// TwinCAT 3 PLC project plc_project
// ProgramVersion: 3.1.4026.24
// libraries:
//   Tc2_Standard, * (Beckhoff Automation GmbH)
//   Tc2_System, * (Beckhoff Automation GmbH)
//   Tc3_Module, * (Beckhoff Automation GmbH)
// project tree:
//   / PlcTask.TcTTO
//   samples/ E_Sample_LargeEnum.TcDUT (not stored), F_Sample_ScaleColorValue.TcPOU (not stored), FB_Sample_AutonomousWarehouseFleetManager.TcPOU, FB_Sample_BatchRecipeExecutionEngine.TcPOU, FB_Sample_DataRingBuffer.TcPOU, FB_Sample_HighDensityDataAnalyticsLogger.TcPOU, FB_Sample_MultiAxisMotionCoordinator.TcPOU (not stored), FB_Sample_MultiStageProcessSupervisor.TcPOU, FB_Sample_StateMachineController.TcPOU (not stored), FB_Sample_ValueBase.TcPOU (not stored), FB_Sample_WidgetBase.TcPOU, GVL_Sample_ParamInflux.TcGVL, GVL_Sample_ShadingConfig.TcGVL (not stored), I_Sample_WidgetInterface.TcIO, ST_Sample_DiagnosticsStruct.TcDUT
//   syntax/ E_Syntax_ExhaustiveComments.TcDUT, E_Syntax_ExplicitIntTyped.TcDUT (not stored), E_Syntax_Flags.TcDUT (not stored), E_Syntax_MultilineAligned.TcDUT (not stored), E_Syntax_TypedExplicit.TcDUT, F_3Args.TcPOU (not stored), F_4Args.TcPOU (not stored), F_5Args.TcPOU (not stored), F_Syntax_Add.TcPOU, F_Syntax_GenericAny.TcPOU, F_Syntax_Return.TcPOU, FB_Syntax_AbstractBase.TcPOU, FB_Syntax_Action.TcPOU (not stored), FB_Syntax_AdvancedSystemExtensions.TcPOU, FB_Syntax_AllVarTypes.TcPOU (not stored), FB_Syntax_AssignAlignmentHeuristics.TcPOU, FB_Syntax_AttributesComprehensive.TcPOU, FB_Syntax_BitAccess.TcPOU, FB_Syntax_Calls.TcPOU (not stored), FB_Syntax_CaseRanges.TcPOU, FB_Syntax_ComplexExpressions.TcPOU, FB_Syntax_ComplexInits.TcPOU, FB_Syntax_ComprehensiveVarBlocks.TcPOU (not stored), FB_Syntax_ConditionalCompile.TcPOU (not stored), FB_Syntax_ControlFlow.TcPOU (not stored), FB_Syntax_DeepControlFlow.TcPOU (not stored), FB_Syntax_DeepNesting.TcPOU, FB_Syntax_Derived.TcPOU, FB_Syntax_DisableRegions.TcPOU (not stored), FB_Syntax_DynamicMem.TcPOU, FB_Syntax_Exceptions.TcPOU (not stored), FB_Syntax_ExhaustiveArraysAndFBInit.TcPOU (not stored), FB_Syntax_ExhaustiveComments.TcPOU, FB_Syntax_ExhaustiveEdgeCases.TcPOU (not stored), FB_Syntax_ExhaustivePragmas.TcPOU (not stored), FB_Syntax_Expressions.TcPOU (not stored), FB_Syntax_ExST.TcPOU, FB_Syntax_FBInitMethods.TcPOU, FB_Syntax_Final.TcPOU (not stored), FB_Syntax_IfMultilineCalls.TcPOU, FB_Syntax_LargeServicePOU.TcPOU, FB_Syntax_LoopControl.TcPOU, FB_Syntax_MathOperators.TcPOU, FB_Syntax_MultiDimArraysAndInits.TcPOU, FB_Syntax_MultiInterfaceDevice.TcPOU (not stored), FB_Syntax_NestedLogCall.TcPOU, FB_Syntax_OOP.TcPOU, FB_Syntax_Pragmas.TcPOU, FB_Syntax_PragmasAndRegions.TcPOU (not stored), FB_Syntax_PropertiesFull.TcPOU, FB_Syntax_PropertySet.TcPOU, FB_Syntax_QueryInterface.TcPOU, FB_Syntax_StringLiterals.TcPOU (not stored), FB_Syntax_StweepDisable.TcPOU, FB_Syntax_SuperThis.TcPOU, FB_Syntax_TimeDate.TcPOU (not stored), FB_Syntax_VarBlocks.TcPOU (not stored), FB_Syntax_VarInOut.TcPOU, FB_Syntax_WrapCallsComprehensive.TcPOU (not stored), FB_Syntax_WrapLongCall.TcPOU, FindAndReplace.TcPOU (not stored), GVL_Syntax_Address.TcGVL, GVL_Syntax_Config.TcGVL (not stored), GVL_Syntax_Global.TcGVL (not stored), GVL_Syntax_Literals.TcGVL, I_Syntax_AdvancedDevice.TcIO (not stored), I_Syntax_BaseDevice.TcIO (not stored), I_Syntax_ExhaustiveComments.TcIO, I_Syntax_Extended.TcIO, I_Syntax_Widget.TcIO (not stored), MAIN.TcPOU, PRG_Syntax_Main.TcPOU, ST_Syntax_Bitfields.TcDUT (not stored), ST_Syntax_ComplexTree.TcDUT (not stored), ST_Syntax_DeepNested.TcDUT (not stored), ST_Syntax_Derived.TcDUT, ST_Syntax_DirectAddressing.TcDUT, ST_Syntax_Dyn.TcDUT (not stored), ST_Syntax_ExhaustiveArrays.TcDUT, ST_Syntax_ExhaustiveComments.TcDUT, ST_Syntax_Mini.TcDUT (not stored), ST_Syntax_PointerRef.TcDUT, T_Syntax_ArraysMultiDim.TcDUT (not stored), T_Syntax_SubrangeEdgeCases.TcDUT, T_Syntax_Types.TcDUT, U_Syntax_ExhaustiveComments.TcDUT, U_Syntax_MultiWordUnion.TcDUT, U_Syntax_Union.TcDUT (not stored)
// real-time tasks:
//   TASK PlcTask: cycle T#10ms, priority 20, ADS port 350

CONFIGURATION plc_project
    RESOURCE PLC ON TwinCAT3
        TASK PlcTask(INTERVAL := T#10ms, PRIORITY := 20);
        PROGRAM MAIN WITH PlcTask : MAIN;
    END_RESOURCE
END_CONFIGURATION

// ---- samples/ST_Sample_DiagnosticsStruct.TcDUT
TYPE ST_Sample_DiagnosticsStruct :
    STRUCT
        (* --- Light device aggregation (previous cycle snapshot) --- *)
        nLightCount                 : UINT; (* Number of reporting light devices *)
        fArtificialLevelSum         : REAL; (* [0..100] - Sum of artificial light levels *)
        fArtificialLevelMean        : REAL; (* [0..100] - Mean artificial light level; 0 if nLightCount = 0 *)
        nLightManualCount           : UINT; (* Number of reporting lights in ManualOperation *)
        nLightExternalOverrideCount : UINT; (* Lights with active prio neither None nor DaylightAutomation *)
        bLightExternalOverride      : BOOL; (* TRUE when nLightExternalOverrideCount > 0 *)
        nLightForeignLightCount     : UINT; (* Of those, the ones actually emitting light (level > 0) *)
        bLightForeignLightActive    : BOOL; (* TRUE when nLightForeignLightCount > 0 *)
        nLightCalibrationCount      : UINT; (* Lights owned by DeskCal this cycle *)

        (* Color temperature aggregation (ColorTemp-capable lights only) *)
        nLightColorTempCount      : UINT; (* Lights reporting a valid color temperature *)
        fLightColorTempKelvinSum  : REAL; (* [K] - Sum of reported color temperatures *)
        fLightColorTempKelvinMean : REAL; (* [K] - Mean color temperature; 0 if nLightColorTempCount = 0 *)

        (* --- Blind device aggregation (previous cycle snapshot) --- *)
        nBlindCount            : UINT; (* Number of reporting blind devices *)
        fBlindPositionSum      : REAL; (* [0..100] - Sum of blind positions *)
        fBlindPositionMean     : REAL; (* [0..100] - Mean blind position; 0 if nBlindCount = 0 *)
        nBlindManualCount      : UINT; (* Number of reporting blinds in ManualOperation *)
        nBlindCalibrationCount : UINT; (* Blinds owned by DeskCal (excl. windows) *)

        (* Angle aggregation (Shade/Sunblind only) *)
        nBlindAngleCount : UINT; (* Blinds reporting a valid angle *)
        fBlindAngleSum   : REAL; (* [deg] - Sum of reported angles *)
        fBlindAngleMean  : REAL; (* [deg] - Mean angle; 0 if nBlindAngleCount = 0 *)

        (* Per NESW facade: 0=North, 1=East, 2=South, 3=West *)
        arrFacadeBlindCount            : ARRAY[0..3] OF UINT; (* Reporting blinds that set this facade bit *)
        arrFacadeBlindPositionMean     : ARRAY[0..3] OF REAL; (* [0..100] - Mean position for that facade bit *)
        arrFacadeBlindCalibrationCount : ARRAY[0..3] OF UINT; (* NESW blinds owned by DeskCal *)
        arrFacadeBlindAngleCount       : ARRAY[0..3] OF UINT; (* Blinds reporting angle for this facade bit *)
        arrFacadeBlindAngleMean        : ARRAY[0..3] OF REAL; (* [deg] - Mean angle for that facade bit *)

        (* --- Occupancy / room sensors (resolved values; *Valid = real source) --- *)
        bMotionSensor              : BOOL; (* Raw motion (sensor or fallback) *)
        bMotionSensorValid         : BOOL; (* TRUE when motion came from stMeasurements *)
        fBrightnessSensorLux       : REAL; (* [Lux] - Effective ceiling / room brightness *)
        bBrightnessSensorValid     : BOOL; (* TRUE when brightness came from stMeasurements *)
        fDeskBrightnessSensorLux   : REAL; (* [Lux] - Effective desk / workplace sensor *)
        bDeskBrightnessSensorValid : BOOL; (* TRUE when desk brightness came from stMeasurements *)
        fHumiditySensor            : REAL; (* [%RH] - Effective room humidity *)
        bHumiditySensorValid       : BOOL; (* TRUE when humidity came from stMeasurements *)
        fCO2Sensor                 : REAL; (* [ppm] - Effective room CO2 / CO2-equivalent *)
        bCO2SensorValid            : BOOL; (* TRUE when CO2 came from stMeasurements *)
        fTemperatureSensor         : REAL; (* [°C] - Effective room temperature *)
        bTemperatureSensorValid    : BOOL; (* TRUE when temperature came from sensor *)
        bOccupancyActive           : BOOL; (* Occupancy: motion hold + Presence delay chains *)
        bOccupancyValid            : BOOL; (* TRUE when occupancy is based on a valid motion sensor *)
    END_STRUCT
END_TYPE

// ---- syntax/E_Syntax_ExhaustiveComments.TcDUT
(*******************************************************************************
 * Enum: E_Syntax_ExhaustiveComments
 * Description: Enumeration with comments on every member and section.
 *******************************************************************************)
TYPE E_Syntax_ExhaustiveComments : (
        // --- Initial / Off states ---
        Uninitialized := 0,  (* System not yet configured *)
        Idle          := 10, // System ready and waiting

        // --- Operational states ---
        Starting := 20, (* Ramping up *)
        Running  := 30, // Normal continuous operation
        Pausing  := 40, (* Transitioning to paused *)
        Paused   := 50, // Temporarily suspended

        // --- Error / Abort states ---
        Stopping      := 80, (* Graceful shutdown *)
        Error         := 90, // Fault detected
        EmergencyStop := 99  (* Immediate safety halt *)
    ) INT;
END_TYPE

// ---- syntax/E_Syntax_TypedExplicit.TcDUT
{attribute 'qualified_only'}
{attribute 'strict'}
TYPE E_Syntax_TypedExplicit : (
        Idle       := 0,   // Initial state
        Starting   := 10,  // Starting sequence
        Running    := 100, // Active processing
        Stopping   := 200, // Ramp down
        ErrorState := -1   // Fault occurred
    ) DINT := Idle;
END_TYPE

// ---- syntax/ST_Syntax_Derived.TcDUT
TYPE ST_Syntax_Derived EXTENDS ST_Syntax_Mini :
    STRUCT
        fExtendedValue : LREAL      := 3.14159;
        sDescription   : STRING(80) := 'Derived Struct';
        bDerivedActive : BOOL;
    END_STRUCT
END_TYPE

// ---- syntax/ST_Syntax_DirectAddressing.TcDUT
TYPE ST_Syntax_DirectAddressing :
    STRUCT
        bInSafetyDoor AT %I* : BOOL;
        nInPosition   AT %I* : INT;
        bOutMotorOn   AT %Q* : BOOL;
        nOutSpeed     AT %Q* : WORD;
        nMemoryStatus AT %M* : DWORD;
    END_STRUCT
END_TYPE

// ---- syntax/ST_Syntax_ExhaustiveArrays.TcDUT
TYPE ST_Syntax_ExhaustiveArrays :
    STRUCT
        arrStaticInts   : ARRAY[1..8] OF INT := [1, 2, 3, 4, 5, 6, 7, 8];
        arrMultiDimInt  : ARRAY[1..2, 1..2] OF INT;
        arrMultilineInt : ARRAY[1..4] OF INT := [
            1, 2,
            3, 4
        ];
        arrNestedMini   : ARRAY[1..2] OF ST_Syntax_Mini := [
            (nId := 1, bActive := TRUE, sName := 'SubA'),
            (nId := 2, bActive := FALSE, sName := 'SubB')
        ];
    END_STRUCT
END_TYPE

// ---- syntax/ST_Syntax_ExhaustiveComments.TcDUT
(*******************************************************************************
 * Struct: ST_Syntax_ExhaustiveComments
 * Description: Data structure with comments in all possible positions.
 *******************************************************************************)
TYPE ST_Syntax_ExhaustiveComments :
    STRUCT
        // --- Identification ---
    nId      : DINT       := 1;      (* Unique device ID *)
        sTag : STRING(31) := 'MAIN'; // System tag name

        // --- Configuration ---
    bEnabled      : BOOL := TRUE;  (* Master enable *)
        fMinLimit : REAL := 0.0;   // Lower threshold
        fMaxLimit : REAL := 100.0; (* Upper threshold *)

        // --- Complex / Nested fields ---
    arrThreshold : ARRAY[1..3] OF REAL := [
        10.0, (* stage 1 *)
        50.0, (* stage 2 *)
        90.0  (* stage 3 *)
    ]; // Multi-stage limits
    END_STRUCT
END_TYPE

// ---- syntax/ST_Syntax_PointerRef.TcDUT
TYPE ST_Syntax_PointerRef :
    STRUCT
        pData : POINTER TO INT;
        rItem : REFERENCE TO INT;
    END_STRUCT
END_TYPE

// ---- syntax/T_Syntax_SubrangeEdgeCases.TcDUT
TYPE T_Syntax_SubrangeEdgeCases : INT(1..100) := 50;

END_TYPE

// ---- syntax/T_Syntax_Types.TcDUT
TYPE T_Syntax_Types :
    STRUCT
        nSubrange   : INT(0..100) := 50;
        aMatrix     : ARRAY[1..3, 1..3] OF REAL;
        sCustomText : STRING(255);
    END_STRUCT
END_TYPE

// ---- syntax/U_Syntax_ExhaustiveComments.TcDUT
(*******************************************************************************
 * Union: U_Syntax_ExhaustiveComments
 * Description: Union testing comments on fields.
 *******************************************************************************)
TYPE U_Syntax_ExhaustiveComments : UNION
        nRawDword : DWORD;               (* 32-bit raw register value *)
        arrBytes  : ARRAY[0..3] OF BYTE; // 4-byte byte access
        arrWords  : ARRAY[0..1] OF WORD; (* 2-word word access *)
    END_UNION
END_TYPE

// ---- syntax/U_Syntax_MultiWordUnion.TcDUT
TYPE U_Syntax_MultiWordUnion : UNION
        nLWord    : LWORD;
        arrDWords : ARRAY[0..1] OF DWORD;
        arrWords  : ARRAY[0..3] OF WORD;
        arrBytes  : ARRAY[0..7] OF BYTE;
    END_UNION
END_TYPE

// ---- samples/GVL_Sample_ParamInflux.TcGVL
{attribute 'qualified_only'}
VAR_GLOBAL CONSTANT
    sDefaultOrg            : STRING(80) := 'ElektroBeckhoff';
    sDefaultBucket         : STRING(80) := 'Telemetry';
    cnMaxBatchSize         : UDINT      := 500;
    cnMaxRetries           : UINT       := 3;
    tDefaultFlushInterval  : TIME       := T#5S;
    tDefaultRequestTimeout : TIME       := T#10S;
END_VAR

// ---- syntax/GVL_Syntax_Address.TcGVL
VAR_GLOBAL
    bInput    AT %I0.0 : BOOL;
    nAnalog   AT %I2   : INT;
    bOutput   AT %Q0.0 : BOOL;
    nSetpoint AT %Q4   : DINT;
END_VAR

// ---- syntax/GVL_Syntax_Literals.TcGVL
VAR_GLOBAL
    todClock           : TOD  := TOD#19:00:00;
    dtEvent            : DT   := DT#2024-01-15-12:30:00;
    nTyped             : DINT := DINT#42;
    nAux, nAux2, nAux3 : UDINT;
END_VAR

// ---- samples/I_Sample_WidgetInterface.TcIO
INTERFACE I_Sample_WidgetInterface EXTENDS __SYSTEM.IQueryInterface

PROPERTY AdsPath : STRING(255)
GET
END_GET
END_PROPERTY

PROPERTY AttributeVariable1 : STRING(80)
GET
END_GET
SET
END_SET
END_PROPERTY

METHOD BuildAttributes : UDINT
VAR_INPUT
    nFlags : DWORD;
END_VAR
END_METHOD

METHOD ProcessCommand : BOOL
VAR_INPUT
    nCommandId : DINT;
    fValue     : LREAL;
END_VAR
VAR_OUTPUT
    bHandled : BOOL;
END_VAR
END_METHOD

END_INTERFACE

// ---- syntax/I_Syntax_ExhaustiveComments.TcIO
(*******************************************************************************
 * Interface: I_Syntax_ExhaustiveComments
 * Description: Interface with doc comments and parameter comments.
 *******************************************************************************)
INTERFACE I_Syntax_ExhaustiveComments EXTENDS __SYSTEM.IQueryInterface

/// <summary>Executes a device command.</summary>
METHOD ExecuteCommand : BOOL
VAR_INPUT
    nCmdId : DINT; (* Command identifier *)
    fParam : LREAL; // Command parameter value
END_VAR
VAR_OUTPUT
    nStatus : UDINT; (* Result status code *)
END_VAR
END_METHOD

/// <summary>True when device is ready.</summary>
PROPERTY P_Operational : BOOL
GET
END_GET
END_PROPERTY

END_INTERFACE

// ---- syntax/I_Syntax_Extended.TcIO
INTERFACE I_Syntax_Extended EXTENDS I_Syntax_Widget

METHOD M_Execute : BOOL
VAR_INPUT
    nCommand : DINT;
END_VAR
END_METHOD

METHOD M_Reset : BOOL
END_METHOD

PROPERTY P_ExtendedStatus : INT
GET
END_GET
END_PROPERTY

END_INTERFACE

// ---- syntax/MAIN.TcPOU
PROGRAM MAIN
VAR
    _nCounter : UDINT;
END_VAR

_nCounter := _nCounter + 1;
PRG_Syntax_Main();

END_PROGRAM

// ---- syntax/PRG_Syntax_Main.TcPOU
PROGRAM PRG_Syntax_Main
VAR
    _nCycle : UDINT;
    _bReady : BOOL;
END_VAR

_nCycle := _nCycle + 1;
_bReady := TRUE;

END_PROGRAM

// ---- samples/FB_Sample_AutonomousWarehouseFleetManager.TcPOU
(*******************************************************************************
 * POU Name:    FB_Sample_AutonomousWarehouseFleetManager
 * Description: Autonomous Mobile Robot (AMR / AGV) warehouse fleet supervisor,
 *              topological 10x10 grid map navigation, A* / Dijkstra pathfinding,
 *              traffic deadlock resolution, dynamic opportunity charging dispatch,
 *              safety laser field scanners, energy feasibility modeling,
 *              methods, actions, and properties (>1000 lines).
 *******************************************************************************)
{attribute 'reflection'}
{attribute 'no_explicit_call' := 'Run cyclic fleet manager via instance call'}
FUNCTION_BLOCK FB_Sample_AutonomousWarehouseFleetManager
VAR_INPUT
    bFleetMasterEnable        : BOOL                := FALSE;   (* Master fleet operations permit *)
    bAutoDispatchEnabled      : BOOL                := TRUE;    (* Autonomous order dispatching active *)
    bForceFleetCharging       : BOOL                := FALSE;   (* Command all idle robots to charge *)
    bEmergencyHaltCommand     : BOOL                := FALSE;   (* Global warehouse emergency stop *)
    bAcknowledgeFleetAlarm    : BOOL                := FALSE;   (* Alarm acknowledgment pulse *)
    bSafetyScannerBypass      : BOOL                := FALSE;   (* Maintenance scanner bypass *)
    nFleetRobotCount          : INT                 := 8;       (* Number of commissioned AGVs [1..16] *)
    nChargingStationCount     : INT                 := 4;       (* Available high-power dock bays *)
    nPriorityQueueLength      : INT                 := 12;      (* Active pending mission backlog *)
    fMinimumBatteryCharge_Pct : REAL                := 25.0;    (* Opportunity charging threshold [%] *)
    fMaxAgvLinearSpeed_mms    : LREAL               := 1200.0;  (* Maximum permissible robot speed [mm/s] *)
    fSafetyZoneClearance_mm   : LREAL               := 350.0;   (* Spatial separation bubble [mm] *)
    tDispatchInterval         : TIME                := T#500MS; (* Order evaluation cycle tick *)
    tHeartbeatTimeout         : TIME                := T#2S;    (* AGV telemetry loss timeout *)
    tChargingSessionDuration  : TIME                := T#3M;    (* Target fast-charge dwell *)
    sWarehouseZoneIdentifier  : STRING(80)          := 'ZONE-LOGISTICS-BAY-4';
    arrChargingStationStatus  : ARRAY[1..4] OF BOOL := [TRUE, TRUE, FALSE, TRUE];
END_VAR
VAR_OUTPUT
    bFleetOperational       : BOOL;        (* High when supervisor is actively routing *)
    bDeadlockDetected       : BOOL;        (* Conflict graph cycle active *)
    bAllRobotsHealthy       : BOOL;        (* High if no AGV reports hardware alarms *)
    bChargingQueueSaturated : BOOL;        (* All charging stations occupied *)
    bGlobalEStopActive      : BOOL;        (* Emergency warehouse halt high *)
    eCurrentFleetPhase      : INT;         (* 0=Idle, 10=OrderIngest, 20=PathPlanning... *)
    nActiveMissionCount     : INT;         (* Currently progressing transport tasks *)
    nTotalFulfilledOrders   : UDINT;       (* Completed warehouse missions counter *)
    nRobotsChargingCount    : INT;         (* AGVs currently docked at chargers *)
    nActiveDeadlockCount    : INT;         (* Resolved traffic deadlocks *)
    fFleetAvailabilityPct   : REAL;        (* Ratio of ready robots [0..100%] *)
    fAverageBatteryLevelPct : REAL;        (* Mean fleet state of charge (SoC) *)
    fGridCongestionIndex    : REAL;        (* Congestion score [0..100%] *)
    nFleetErrorCode         : UDINT;       (* 0=OK, 16#C001=Deadlock, 16#C002=LostHeartbeat *)
    sDetailedFleetStatus    : STRING(255); (* Operator readable diagnostic line *)
    tExecutionTimeInPhase   : TIME;        (* Phase execution stopwatch *)
END_VAR
VAR_IN_OUT
    stDiagnostics : ST_Sample_DiagnosticsStruct; (* Shared plant diagnostic bus *)
END_VAR
VAR
    // --- 1. Subordinate Function Blocks and Timers ---
    _fbFleetStateController   : FB_Sample_StateMachineController;
    _fbMissionQueueBuffer     : FB_Sample_DataRingBuffer;
    _fbRTrigDispatch          : R_TRIG;
    _fbRTrigCharge            : R_TRIG;
    _fbRTrigEStop             : R_TRIG;
    _fbRTrigAckAlarm          : R_TRIG;
    _fbTonDispatchTicker      : TON;
    _fbTonHeartbeatWatchdog   : TON;
    _fbTonDeadlockSettleTimer : TON;
    _fbTonChargingDwellTimer  : TON;

    // --- 2. State Machine Engine Registers ---
    _nMasterFleetState        : INT  := 0;     (* Master fleet supervisor sequence index *)
    _nPreviousFleetState      : INT  := 0;     (* Saved state prior to halt *)
    _nOrderBacklogIndex       : INT  := 0;     (* Active order iterator *)
    _nRetryRoutingAttempts    : INT  := 0;     (* A* path retry counter *)
    _bSafetyLaserFieldTripped : BOOL := FALSE; (* Spatial optical scanner trip *)
    _bDeadlockResolverActive  : BOOL := FALSE; (* Deadlock unblock in progress *)

    // --- 3. AGV Telemetry, Position and Battery Arrays ---
    _arrAgvCurrentX_mm      : ARRAY[1..16] OF LREAL; (* Odometry X coordinate *)
    _arrAgvCurrentY_mm      : ARRAY[1..16] OF LREAL; (* Odometry Y coordinate *)
    _arrAgvTargetNodeX      : ARRAY[1..16] OF INT;   (* Target topological node X [1..10] *)
    _arrAgvTargetNodeY      : ARRAY[1..16] OF INT;   (* Target topological node Y [1..10] *)
    _arrAgvBatterySoC_Pct   : ARRAY[1..16] OF REAL;
    _arrAgvStateCodes       : ARRAY[1..16] OF INT;  (* 0=Idle, 1=InTransit, 2=Docking, 3=Charging *)
    _arrAgvHeartbeatMissing : ARRAY[1..16] OF BOOL; (* Communications loss flags *)

    // --- 4. 10x10 Topological Grid Cost & Occupancy Map ---
    _arrTopologicalGridMap   : ARRAY[1..10, 1..10] OF INT := [
        1, 1, 1, 1, 5, 1, 1, 1, 1, 1,
        1, 9, 9, 1, 5, 1, 9, 9, 1, 1,
        1, 9, 9, 1, 1, 1, 9, 9, 1, 1,
        1, 1, 1, 1, 1, 1, 1, 1, 1, 1,
        5, 5, 1, 9, 9, 9, 9, 1, 5, 5,
        5, 5, 1, 9, 9, 9, 9, 1, 5, 5,
        1, 1, 1, 1, 1, 1, 1, 1, 1, 1,
        1, 9, 9, 1, 1, 1, 9, 9, 1, 1,
        1, 9, 9, 1, 5, 1, 9, 9, 1, 1,
        1, 1, 1, 1, 5, 1, 1, 1, 1, 1
    ];
    _arrNodeOccupancyMatrix : ARRAY[1..10, 1..10] OF INT; (* ID of AGV occupying node (0=Empty) *)
    _arrMissionPriorityList : ARRAY[1..16] OF INT := [1, 3, 2, 4, 1, 2, 1, 3, 2, 1, 4, 2, 1, 3, 2, 1];

    // --- 5. Internal Strings and Diagnostic Text ---
    _sActiveFleetPhaseName  : STRING(80) := 'STANDBY_IDLE';
    _sFleetAuditSummary     : STRING(255);
    _sLatestMissionDispatch : STRING(80) := 'NO_MISSION_DISPATCHED';
END_VAR
VAR_TEMP
    _nTempAgvIdx           : INT;
    _nTempGridX            : INT;
    _nTempGridY            : INT;
    _fTempBatterySum       : REAL;
    _fTempDistDelta        : LREAL;
    _bTempPathPlanningOk   : BOOL;
    _bTempConflictResolved : BOOL;
END_VAR
VAR CONSTANT
    cMaxWarehouseFleetSize   : INT   := 16;
    cGridDimensionNodes      : INT   := 10;
    cNodeSpacing_mm          : LREAL := 1000.0;
    cCriticalLowBatteryLevel : REAL  := 15.0;
    cObstacleNodeWeight      : INT   := 9;
END_VAR

// =============================================================================
// 1. SIGNAL INGESTION, OPERATOR COMMANDS & SAFETY FIELDS
// =============================================================================
{region "Warehouse Fleet Safety & Interlocks"}
    _fbRTrigDispatch(CLK := bAutoDispatchEnabled);
    _fbRTrigCharge(CLK := bForceFleetCharging);
    _fbRTrigEStop(CLK := bEmergencyHaltCommand);
    _fbRTrigAckAlarm(CLK := bAcknowledgeFleetAlarm);

    // Reset alarm latch on operator pulse
    IF _fbRTrigAckAlarm.Q THEN
        bDeadlockDetected     := FALSE;
        bGlobalEStopActive    := FALSE;
        nFleetErrorCode       := 0;
        sDetailedFleetStatus  := 'Fleet alarms cleared by operator.';
END_IF

    // Emergency halt forces immediate fleet standstill
    IF _fbRTrigEStop.Q OR (bFleetMasterEnable = FALSE AND _nMasterFleetState > 0) THEN
        _nMasterFleetState    := 900; // Global E-Stop
        bGlobalEStopActive    := TRUE;
        sDetailedFleetStatus  := 'GLOBAL WAREHOUSE EMERGENCY HALT TRIGGERED!';
END_IF

    // Periodic dispatch evaluation ticker
    _fbTonDispatchTicker(IN := NOT _fbTonDispatchTicker.Q, PT := tDispatchInterval);

    IF _fbTonDispatchTicker.Q AND bFleetMasterEnable THEN
        A_ScanSafetyFieldSensors();
        A_UpdateWarehouseFleetKPIs();
        A_BroadcastFleetHeartbeat();
        A_EvaluateEmergencyEStopConditions();
        A_BroadcastSafetyScannerFields();
        A_UpdateWarehouseThroughputMetrics();
END_IF

    // Heartbeat loss watchdog
    _fbTonHeartbeatWatchdog(IN := (_nMasterFleetState > 0 AND _nMasterFleetState < 800), PT := tHeartbeatTimeout);

    IF _fbTonHeartbeatWatchdog.Q AND NOT bDeadlockDetected THEN
        FOR _nTempAgvIdx := 1 TO nFleetRobotCount DO
            IF _arrAgvHeartbeatMissing[_nTempAgvIdx] THEN
                bAllRobotsHealthy := FALSE;
                nFleetErrorCode      := 16#C002; // Missing heartbeat
                sDetailedFleetStatus := 'FAULT: Lost telemetry heartbeat from one or more AGVs!';
        END_IF
        END_FOR
END_IF
{endregion}

// =============================================================================
// 2. MASTER WAREHOUSE FLEET ORCHESTRATION (10-STATE ENGINE)
// =============================================================================
CASE _nMasterFleetState OF

    0:
        // STATE 0: IDLE STANDBY
        _sActiveFleetPhaseName := 'STANDBY_IDLE';
        bFleetOperational      := FALSE;
        bDeadlockDetected      := FALSE;
        nActiveMissionCount    := 0;
        nRobotsChargingCount   := 0;

        IF bFleetMasterEnable AND NOT bGlobalEStopActive THEN
            _nMasterFleetState   := 10; // Proceed to Order Ingestion
            bFleetOperational    := TRUE;
            sDetailedFleetStatus := 'Fleet supervisor operational. Ingesting transport orders.';
        END_IF

    10:
        // STATE 10: INGEST & PRIORITIZE TRANSPORT ORDERS
        _sActiveFleetPhaseName := 'ORDER_INGESTION_AND_PRIORITY';

        M_SortPriorityOrderQueue(arrPriorities := _arrMissionPriorityList, nQueueLen := nPriorityQueueLength);

        _nMasterFleetState   := 20; // Proceed to Topological A* Path Planning
        sDetailedFleetStatus := 'Orders prioritized. Planning topological collision-free routes.';

    20:
        // STATE 20: TOPOLOGICAL A* SHORTEST ROUTE PLANNING
        _sActiveFleetPhaseName := 'TOPOLOGICAL_ASTAR_ROUTING';

        _bTempPathPlanningOk := M_PlanAStarTopologicalRoute(nStartNodeX := 1, nStartNodeY := 1, nGoalNodeX := 10, nGoalNodeY := 10);

        IF _bTempPathPlanningOk THEN
            _nMasterFleetState   := 30; // Proceed to Traffic Conflict Negotiation
            sDetailedFleetStatus := 'Topological paths calculated. Negotiating spatial reservations.';
        ELSE
            _nRetryRoutingAttempts := _nRetryRoutingAttempts + 1;

            IF _nRetryRoutingAttempts > 3 THEN
                nFleetErrorCode      := 16#C020;
                sDetailedFleetStatus := 'Routing failed: Target node unreachable due to map obstacles!';
                _nMasterFleetState   := 70; // Attempt deadlock unblock
            END_IF
        END_IF

    30:
        // STATE 30: MULTI-AGENT TRAFFIC CONFLICT NEGOTIATION
        _sActiveFleetPhaseName := 'TRAFFIC_CONFLICT_NEGOTIATION';

        _bTempConflictResolved := M_ResolveFleetTrafficDeadlock();

        IF _bTempConflictResolved THEN
            _nMasterFleetState   := 40; // Proceed to Mission Dispatch
            sDetailedFleetStatus := 'Spatial conflicts cleared. Dispatching tasks to robot fleet.';
        ELSE
            bDeadlockDetected := TRUE;
            _nMasterFleetState   := 70; // Deadlock resolution state
            sDetailedFleetStatus := 'Traffic conflict detected: Negotiating wait points.';
        END_IF

    40:
        // STATE 40: MISSION DISPATCH & AGV TASK COMMITMENT
        _sActiveFleetPhaseName := 'MISSION_DISPATCH_COMMIT';

        FOR _nTempAgvIdx := 1 TO nFleetRobotCount DO
            IF _arrAgvStateCodes[_nTempAgvIdx] = 0 THEN // If AGV is Idle
                IF _arrAgvBatterySoC_Pct[_nTempAgvIdx] < fMinimumBatteryCharge_Pct THEN
                    _arrAgvStateCodes[_nTempAgvIdx] := 3; // Send to Charging
                ELSE
                    M_AssignTransportMissionOrder(nRobotId := _nTempAgvIdx, nTargetX := 8, nTargetY := 8, nPriority := 2);
                    _arrAgvStateCodes[_nTempAgvIdx] := 1; // In Transit
                    nActiveMissionCount := nActiveMissionCount + 1;
                END_IF
            END_IF
        END_FOR

        _nMasterFleetState   := 50; // Proceed to Real-Time Monitoring
        sDetailedFleetStatus := 'Missions dispatched. Monitoring odometry and safety fields.';

    50:
        // STATE 50: REAL-TIME FLEET TELEMETRY & ODOMETRY TRACKING
        _sActiveFleetPhaseName := 'REALTIME_FLEET_TRACKING';

        FOR _nTempAgvIdx := 1 TO nFleetRobotCount DO
            IF _arrAgvStateCodes[_nTempAgvIdx] = 1 THEN
                // Simulate incremental robot motion towards goal node
                _arrAgvCurrentX_mm[_nTempAgvIdx] := _arrAgvCurrentX_mm[_nTempAgvIdx] + 25.0;
                IF _arrAgvCurrentX_mm[_nTempAgvIdx] >= (TO_LREAL(_arrAgvTargetNodeX[_nTempAgvIdx]) * cNodeSpacing_mm) THEN
                    _arrAgvStateCodes[_nTempAgvIdx] := 0; // Mission Finished
                    nActiveMissionCount   := nActiveMissionCount - 1;
                    nTotalFulfilledOrders := nTotalFulfilledOrders + 1;
                END_IF
            END_IF
        END_FOR

        IF bForceFleetCharging THEN
            _nMasterFleetState   := 60; // Advance to Charging Balancing
            sDetailedFleetStatus := 'Operator forced fleet charging cycle.';
        ELSIF nActiveMissionCount = 0 THEN
            _nMasterFleetState   := 100; // All Active Orders Fulfilled
            sDetailedFleetStatus := 'Active mission backlog complete. Returning to standby.';
        END_IF

    60:
        // STATE 60: OPPORTUNITY BATTERY BALANCING & CHARGING DOCKING
        _sActiveFleetPhaseName := 'BATTERY_BALANCING_CHARGING';

        M_OptimizeFleetBatteryCharging(arrChargerStatus := arrChargingStationStatus, arrSoC_Pct := _arrAgvBatterySoC_Pct);

        _fbTonChargingDwellTimer(IN := TRUE, PT := tChargingSessionDuration);

        IF _fbTonChargingDwellTimer.Q THEN
            _fbTonChargingDwellTimer(IN := FALSE);
            _nMasterFleetState   := 10; // Return to Order Ingestion
            sDetailedFleetStatus := 'Charging cycle completed. Ready for next transport orders.';
        END_IF

    70:
        // STATE 70: DEADLOCK RESOLUTION & DYNAMIC REROUTING
        _sActiveFleetPhaseName := 'DEADLOCK_REROUTING_RESOLVER';

        _fbTonDeadlockSettleTimer(IN := TRUE, PT := T#1S);

        IF _fbTonDeadlockSettleTimer.Q THEN
            _fbTonDeadlockSettleTimer(IN := FALSE);
            bDeadlockDetected    := FALSE;
            nActiveDeadlockCount := nActiveDeadlockCount + 1;
            _nMasterFleetState   := 20; // Re-plan routes
            sDetailedFleetStatus := 'Deadlock resolved via lower priority AGV backoff.';
        END_IF

    100:
        // STATE 100: FLEET MISSION BATCH COMPLETED
        _sActiveFleetPhaseName := 'MISSION_BATCH_COMPLETED';
        bFleetOperational      := TRUE;

        M_FormatFleetStatusJSON(sZoneTag := sWarehouseZoneIdentifier);

        _nMasterFleetState   := 0; // Return to Standby
        sDetailedFleetStatus := 'Fleet orders fulfilled successfully.';

    800:
        // STATE 800: FAULT STATE & SAFETY FIELD INTERRUPT
        _sActiveFleetPhaseName := 'FAULT_SAFETY_LOCKDOWN';
        bFleetOperational      := FALSE;

        IF _fbRTrigAckAlarm.Q AND nFleetErrorCode = 0 THEN
            _nMasterFleetState   := 0;
            sDetailedFleetStatus := 'Fault cleared. Supervisor returned to standby.';
        END_IF

    900:
        // STATE 900: GLOBAL WAREHOUSE EMERGENCY HALT
        _sActiveFleetPhaseName := 'GLOBAL_EMERGENCY_HALT';
        M_TriggerEmergencyWarehouseHalt();

        IF _fbRTrigAckAlarm.Q THEN
            bGlobalEStopActive := FALSE;
            _nMasterFleetState   := 800; // Transition to Fault State
            sDetailedFleetStatus := 'Emergency stop reset. Awaiting supervisor clearance.';
        END_IF

ELSE
    _nMasterFleetState   := 800;
    nFleetErrorCode      := 16#C999;
    sDetailedFleetStatus := 'FATAL: Unknown fleet supervisor state index encountered.';
END_CASE

eCurrentFleetPhase    := _nMasterFleetState;
fFleetAvailabilityPct := M_CalculateFleetAvailabilityIndex();

ACTION A_BroadcastFleetHeartbeat:
// Periodic heartbeat ping to central SCADA
stDiagnostics.fDeskBrightnessSensorLux := TO_REAL(nTotalFulfilledOrders);
END_ACTION

ACTION A_BroadcastSafetyScannerFields:
// Safety field scanner heartbeat
IF NOT bSafetyScannerBypass THEN
    stDiagnostics.nLightCount := stDiagnostics.nLightCount + 1;
END_IF
END_ACTION

ACTION A_EvaluateEmergencyEStopConditions:
// Check if all robots are safe
IF _bSafetyLaserFieldTripped AND NOT bSafetyScannerBypass THEN
    _nMasterFleetState := 900;
END_IF
END_ACTION

ACTION A_ScanSafetyFieldSensors:
// Optical safety field area scan
_bSafetyLaserFieldTripped := FALSE;

FOR _nTempAgvIdx := 1 TO nFleetRobotCount DO
    IF _arrAgvBatterySoC_Pct[_nTempAgvIdx] <= cCriticalLowBatteryLevel THEN
        _arrAgvStateCodes[_nTempAgvIdx] := 3; // Force to charger
    END_IF
END_FOR
END_ACTION

ACTION A_UpdateWarehouseFleetKPIs:
// Calculate mean battery level across all robots
_fTempBatterySum := 0.0;

FOR _nTempAgvIdx := 1 TO nFleetRobotCount DO
    _fTempBatterySum := _fTempBatterySum + _arrAgvBatterySoC_Pct[_nTempAgvIdx];
END_FOR

IF nFleetRobotCount > 0 THEN
    fAverageBatteryLevelPct := _fTempBatterySum / TO_REAL(nFleetRobotCount);
END_IF

// Update diagnostic interface bus
stDiagnostics.nLightCount         := TO_UINT(nFleetRobotCount);
stDiagnostics.fArtificialLevelSum := fAverageBatteryLevelPct;
END_ACTION

ACTION A_UpdateWarehouseThroughputMetrics:
// Compute hourly throughput estimate
stDiagnostics.fBlindPositionSum := TO_REAL(nTotalFulfilledOrders * 12);
END_ACTION

METHOD M_AssignTransportMissionOrder : BOOL
VAR_INPUT
    nRobotId  : INT;
    nTargetX  : INT;
    nTargetY  : INT;
    nPriority : INT;
END_VAR
IF nRobotId >= 1 AND nRobotId <= 16 THEN
    _arrAgvTargetNodeX[nRobotId]  := nTargetX;
    _arrAgvTargetNodeY[nRobotId]  := nTargetY;
    _sLatestMissionDispatch       := CONCAT('ORDER_DISPATCHED_TO_AGV_', INT_TO_STRING(nRobotId));
    M_AssignTransportMissionOrder := TRUE;
ELSE
    M_AssignTransportMissionOrder := FALSE;
END_IF
END_METHOD

METHOD M_CalculateFleetAvailabilityIndex : REAL
VAR
    _nIdx   : INT;
    _nReady : INT := 0;
END_VAR
FOR _nIdx := 1 TO nFleetRobotCount DO
    IF _arrAgvStateCodes[_nIdx] = 0 OR _arrAgvStateCodes[_nIdx] = 1 THEN
        _nReady := _nReady + 1;
    END_IF
END_FOR

IF nFleetRobotCount > 0 THEN
    M_CalculateFleetAvailabilityIndex := (TO_REAL(_nReady) / TO_REAL(nFleetRobotCount)) * 100.0;
ELSE
    M_CalculateFleetAvailabilityIndex := 0.0;
END_IF
END_METHOD

METHOD M_CalculateFleetMissionEfficiency : REAL
VAR_INPUT
    fTotalEnergyConsumedKWh  : REAL;
    fTotalDistanceTraveledKm : REAL;
END_VAR
IF fTotalDistanceTraveledKm > 0.0 THEN
    M_CalculateFleetMissionEfficiency := fTotalEnergyConsumedKWh / fTotalDistanceTraveledKm;
ELSE
    M_CalculateFleetMissionEfficiency := 0.0;
END_IF
END_METHOD

METHOD M_CalculateFleetTurnaroundTime : LREAL
VAR_INPUT
    fAverageDistanceM : LREAL;
    fAverageSpeedMms  : LREAL;
END_VAR
IF fAverageSpeedMms > 0.0 THEN
    M_CalculateFleetTurnaroundTime := (fAverageDistanceM * 1000.0) / fAverageSpeedMms;
ELSE
    M_CalculateFleetTurnaroundTime := 0.0;
END_IF
END_METHOD

METHOD M_CalculateManhattanDistance : LREAL
VAR_INPUT
    nX1 : INT;
    nY1 : INT;
    nX2 : INT;
    nY2 : INT;
END_VAR
M_CalculateManhattanDistance := TO_LREAL(ABS(nX1 - nX2) + ABS(nY1 - nY2));
END_METHOD

METHOD M_CalibrateFloorGridCoordinates : BOOL
VAR_INPUT
    nGridOriginX_mm : LREAL;
    nGridOriginY_mm : LREAL;
END_VAR
M_CalibrateFloorGridCoordinates := (nGridOriginX_mm >= 0.0 AND nGridOriginY_mm >= 0.0);
END_METHOD

METHOD M_ComputeDynamicNodeCosts : BOOL
VAR
    _nX : INT;
    _nY : INT;
END_VAR
FOR _nX := 1 TO 10 DO
    FOR _nY := 1 TO 10 DO
        IF _arrNodeOccupancyMatrix[_nX, _nY] > 0 THEN
            _arrTopologicalGridMap[_nX, _nY] := 8; // Heavy penalty on occupied cells
        ELSIF _arrTopologicalGridMap[_nX, _nY] <> 9 THEN
            _arrTopologicalGridMap[_nX, _nY] := 1; // Default low travel cost
        END_IF
    END_FOR
END_FOR

M_ComputeDynamicNodeCosts := TRUE;
END_METHOD

METHOD M_EstimateMissionEnergyFeasibility : BOOL
VAR_INPUT
    nRobotId     : INT;
    fDistance_m  : LREAL;
    fPayloadMass : REAL;
END_VAR
VAR
    _fEnergyRequiredPct : REAL;
END_VAR
IF nRobotId < 1 OR nRobotId > 16 THEN
    M_EstimateMissionEnergyFeasibility := FALSE;
    RETURN;
END_IF

_fEnergyRequiredPct                := TO_REAL(fDistance_m * 0.05) * (1.0 + (fPayloadMass * 0.01));
M_EstimateMissionEnergyFeasibility := (_arrAgvBatterySoC_Pct[nRobotId] > (_fEnergyRequiredPct + fMinimumBatteryCharge_Pct));
END_METHOD

METHOD M_EvaluateInterRobotClearance : BOOL
VAR_INPUT
    nRobotA : INT;
    nRobotB : INT;
END_VAR
VAR
    _fDX   : LREAL;
    _fDY   : LREAL;
    _fDist : LREAL;
END_VAR
IF nRobotA < 1 OR nRobotA > 16 OR nRobotB < 1 OR nRobotB > 16 THEN
    M_EvaluateInterRobotClearance := FALSE;
    RETURN;
END_IF

_fDX   := _arrAgvCurrentX_mm[nRobotA] - _arrAgvCurrentX_mm[nRobotB];
_fDY   := _arrAgvCurrentY_mm[nRobotA] - _arrAgvCurrentY_mm[nRobotB];
_fDist := SQRT((_fDX * _fDX) + (_fDY * _fDY));

M_EvaluateInterRobotClearance := (_fDist >= fSafetyZoneClearance_mm);
END_METHOD

METHOD M_EvaluateNodeOccupancyRisk : INT
VAR_INPUT
    nNodeX : INT;
    nNodeY : INT;
END_VAR
IF nNodeX >= 1 AND nNodeX <= 10 AND nNodeY >= 1 AND nNodeY <= 10 THEN
    M_EvaluateNodeOccupancyRisk := _arrTopologicalGridMap[nNodeX, nNodeY];
ELSE
    M_EvaluateNodeOccupancyRisk := 99;
END_IF
END_METHOD

METHOD M_FindNearestAvailableChargingBay : INT
VAR_INPUT
    fRobotX : LREAL;
    fRobotY : LREAL;
END_VAR
VAR
    _nIdx : INT;
END_VAR
FOR _nIdx := 1 TO 4 DO
    IF arrChargingStationStatus[_nIdx] THEN
        M_FindNearestAvailableChargingBay := _nIdx;
        RETURN;
    END_IF
END_FOR

M_FindNearestAvailableChargingBay := 0;
END_METHOD

METHOD M_FormatAgvStatusReport : STRING(255)
VAR_INPUT
    nRobotId : INT;
END_VAR
VAR
    _sResult : STRING(255);
    _sId     : STRING(10);
    _sSoC    : STRING(20);
END_VAR
IF nRobotId < 1 OR nRobotId > 16 THEN
    M_FormatAgvStatusReport := 'INVALID_ROBOT_ID';
    RETURN;
END_IF

_sId  := INT_TO_STRING(nRobotId);
_sSoC := REAL_TO_STRING(_arrAgvBatterySoC_Pct[nRobotId]);

_sResult := CONCAT('AGV_ID: ', _sId);
_sResult := CONCAT(_sResult, ' | SoC: ');
_sResult := CONCAT(_sResult, _sSoC);
_sResult := CONCAT(_sResult, '% | State: ACTIVE');

M_FormatAgvStatusReport := _sResult;
END_METHOD

METHOD M_FormatFleetStatusJSON : STRING(255)
VAR_INPUT
    sZoneTag : STRING(50);
END_VAR
VAR
    _sResult   : STRING(255);
    _sMissions : STRING(10);
    _sRobots   : STRING(10);
END_VAR
_sMissions := INT_TO_STRING(nActiveMissionCount);
_sRobots   := INT_TO_STRING(nFleetRobotCount);

_sResult := CONCAT('{"zone":"', sZoneTag);
_sResult := CONCAT(_sResult, '","active_missions":');
_sResult := CONCAT(_sResult, _sMissions);
_sResult := CONCAT(_sResult, ',"fleet_size":');
_sResult := CONCAT(_sResult, _sRobots);
_sResult := CONCAT(_sResult, ',"status":"OPERATIONAL"}');

_sFleetAuditSummary     := _sResult;
M_FormatFleetStatusJSON := _sResult;
END_METHOD

METHOD M_HeuristicEuclideanCost : LREAL
VAR_INPUT
    nX1 : INT;
    nY1 : INT;
    nX2 : INT;
    nY2 : INT;
END_VAR
VAR
    _fDX : LREAL;
    _fDY : LREAL;
END_VAR
_fDX := TO_LREAL(nX1 - nX2);
_fDY := TO_LREAL(nY1 - nY2);

M_HeuristicEuclideanCost := SQRT((_fDX * _fDX) + (_fDY * _fDY));
END_METHOD

METHOD M_OptimizeFleetBatteryCharging : BOOL
VAR_INPUT
    arrChargerStatus : ARRAY[1..4] OF BOOL;
    arrSoC_Pct       : ARRAY[1..16] OF REAL;
END_VAR
VAR
    _nRobotIdx : INT;
    _nDockIdx  : INT;
END_VAR
nRobotsChargingCount := 0;

FOR _nRobotIdx := 1 TO nFleetRobotCount DO
    IF arrSoC_Pct[_nRobotIdx] < fMinimumBatteryCharge_Pct THEN
        FOR _nDockIdx := 1 TO 4 DO
            IF arrChargerStatus[_nDockIdx] THEN
                _arrAgvStateCodes[_nRobotIdx] := 3; // Docked and charging
                nRobotsChargingCount := nRobotsChargingCount + 1;
                EXIT;
            END_IF
        END_FOR
    END_IF
END_FOR

M_OptimizeFleetBatteryCharging := (nRobotsChargingCount > 0);
END_METHOD

METHOD M_PlanAStarTopologicalRoute : BOOL
VAR_INPUT
    nStartNodeX : INT;
    nStartNodeY : INT;
    nGoalNodeX  : INT;
    nGoalNodeY  : INT;
END_VAR
VAR
    _fH : LREAL;
END_VAR
IF nStartNodeX < 1 OR nStartNodeX > 10 OR nGoalNodeX < 1 OR nGoalNodeX > 10 THEN
    M_PlanAStarTopologicalRoute := FALSE;
    RETURN;
END_IF

_fH := M_HeuristicEuclideanCost(nX1 := nStartNodeX, nY1 := nStartNodeY, nX2 := nGoalNodeX, nY2 := nGoalNodeY);

M_PlanAStarTopologicalRoute := (_fH < 100.0);
END_METHOD

METHOD M_PreconditionBatteryThermals : BOOL
VAR_INPUT
    nRobotId : INT;
END_VAR
IF nRobotId >= 1 AND nRobotId <= 16 THEN
    // Active cooling fan permit on rapid charge
    M_PreconditionBatteryThermals := (_arrAgvBatterySoC_Pct[nRobotId] < 80.0);
ELSE
    M_PreconditionBatteryThermals := FALSE;
END_IF
END_METHOD

METHOD M_ProcessAgvHeartbeatPacket : BOOL
VAR_INPUT
    nRobotId    : INT;
    fX_mm       : LREAL;
    fY_mm       : LREAL;
    fBatterySoC : REAL;
END_VAR
IF nRobotId >= 1 AND nRobotId <= 16 THEN
    _arrAgvCurrentX_mm[nRobotId]      := fX_mm;
    _arrAgvCurrentY_mm[nRobotId]      := fY_mm;
    _arrAgvBatterySoC_Pct[nRobotId]   := fBatterySoC;
    _arrAgvHeartbeatMissing[nRobotId] := FALSE;
    M_ProcessAgvHeartbeatPacket       := TRUE;
ELSE
    M_ProcessAgvHeartbeatPacket := FALSE;
END_IF
END_METHOD

METHOD M_ResolveFleetTrafficDeadlock : BOOL
VAR
    _nIdxA : INT;
    _nIdxB : INT;
    _fDist : LREAL;
END_VAR
FOR _nIdxA := 1 TO nFleetRobotCount DO
    FOR _nIdxB := _nIdxA + 1 TO nFleetRobotCount DO
        _fDist := M_CalculateManhattanDistance(
                nX1 := TO_INT(_arrAgvCurrentX_mm[_nIdxA] / 1000.0),
                nY1 := TO_INT(_arrAgvCurrentY_mm[_nIdxA] / 1000.0),
                nX2 := TO_INT(_arrAgvCurrentX_mm[_nIdxB] / 1000.0),
                nY2 := TO_INT(_arrAgvCurrentY_mm[_nIdxB] / 1000.0));

        IF _fDist < 1.0 THEN
            // Yield priority to lower index AGV
            _arrAgvStateCodes[_nIdxB]     := 0;
            M_ResolveFleetTrafficDeadlock := FALSE;
            RETURN;
        END_IF
    END_FOR
END_FOR

M_ResolveFleetTrafficDeadlock := TRUE;
END_METHOD

METHOD M_SortPriorityOrderQueue : BOOL
VAR_INPUT
    arrPriorities : ARRAY[1..16] OF INT;
    nQueueLen     : INT;
END_VAR
VAR
    _i    : INT;
    _j    : INT;
    _temp : INT;
END_VAR
IF nQueueLen > 16 THEN
    M_SortPriorityOrderQueue := FALSE;
    RETURN;
END_IF

FOR _i := 1 TO nQueueLen - 1 DO
    FOR _j := 1 TO nQueueLen - _i DO
        IF _arrMissionPriorityList[_j] < _arrMissionPriorityList[_j + 1] THEN
            _temp                           := _arrMissionPriorityList[_j];
            _arrMissionPriorityList[_j]     := _arrMissionPriorityList[_j + 1];
            _arrMissionPriorityList[_j + 1] := _temp;
        END_IF
    END_FOR
END_FOR

M_SortPriorityOrderQueue := TRUE;
END_METHOD

METHOD M_TriggerEmergencyWarehouseHalt : BOOL
VAR
    _nIdx : INT;
END_VAR
FOR _nIdx := 1 TO 16 DO
    _arrAgvStateCodes[_nIdx] := 0; // Force immediate standstill
END_FOR

M_TriggerEmergencyWarehouseHalt := TRUE;
END_METHOD

PROPERTY P_ActiveGridCongestionScore : REAL
GET
P_ActiveGridCongestionScore := (TO_REAL(nActiveMissionCount) / TO_REAL(cGridDimensionNodes)) * 100.0;
END_GET
END_PROPERTY

PROPERTY P_ActiveMissionQueueLength : INT
GET
P_ActiveMissionQueueLength := nActiveMissionCount;
END_GET
END_PROPERTY

PROPERTY P_ActiveTrafficReservationCount : INT
GET
P_ActiveTrafficReservationCount := nActiveMissionCount;
END_GET
END_PROPERTY

PROPERTY P_FleetAvailabilityRatio : REAL
GET
P_FleetAvailabilityRatio := fFleetAvailabilityPct;
END_GET
END_PROPERTY

PROPERTY P_FleetChargingThreshold : REAL
GET
P_FleetChargingThreshold := fMinimumBatteryCharge_Pct;
END_GET
SET
IF P_FleetChargingThreshold >= 10.0 AND P_FleetChargingThreshold <= 50.0 THEN
    fMinimumBatteryCharge_Pct := P_FleetChargingThreshold;
END_IF
END_SET
END_PROPERTY

PROPERTY P_FleetEnergyStateOfCharge : REAL
GET
P_FleetEnergyStateOfCharge := fAverageBatteryLevelPct;
END_GET
SET
fAverageBatteryLevelPct := P_FleetEnergyStateOfCharge;
END_SET
END_PROPERTY

PROPERTY P_FleetSafetyEnvelopeMargin : LREAL
GET
P_FleetSafetyEnvelopeMargin := fSafetyZoneClearance_mm;
END_GET
END_PROPERTY

PROPERTY P_TotalFulfilledMissions : UDINT
GET
P_TotalFulfilledMissions := nTotalFulfilledOrders;
END_GET
END_PROPERTY

END_FUNCTION_BLOCK

// ---- samples/FB_Sample_DataRingBuffer.TcPOU
FUNCTION_BLOCK FB_Sample_DataRingBuffer
VAR CONSTANT
    cBufferSize : INT := 64;
END_VAR
VAR_OUTPUT
    nCount : INT;
    bFull  : BOOL;
    bEmpty : BOOL := TRUE;
END_VAR
VAR
    _arrBuffer : ARRAY[0..63] OF LREAL;
    _nHead     : INT;
    _nTail     : INT;
    _nCount    : INT;
END_VAR

nCount := _nCount;
bEmpty := (_nCount = 0);
bFull  := (_nCount >= cBufferSize);

METHOD M_Clear : BOOL
_nHead  := 0;
_nTail  := 0;
_nCount := 0;
M_Clear := TRUE;
END_METHOD

METHOD M_Pop : BOOL
VAR_OUTPUT
    fValue : LREAL;
END_VAR
IF _nCount <= 0 THEN
    fValue := 0.0;
    M_Pop  := FALSE;
    RETURN;
END_IF

fValue  := _arrBuffer[_nTail];
_nTail  := (_nTail + 1) MOD cBufferSize;
_nCount := _nCount - 1;
M_Pop   := TRUE;
END_METHOD

METHOD M_Push : BOOL
VAR_INPUT
    fValue : LREAL;
END_VAR
IF _nCount >= cBufferSize THEN
    M_Push := FALSE;
    RETURN;
END_IF

_arrBuffer[_nHead] := fValue;
_nHead             := (_nHead + 1) MOD cBufferSize;
_nCount            := _nCount + 1;
M_Push             := TRUE;
END_METHOD

END_FUNCTION_BLOCK

// ---- samples/FB_Sample_BatchRecipeExecutionEngine.TcPOU
(*******************************************************************************
 * POU Name:    FB_Sample_BatchRecipeExecutionEngine
 * Description: Massive multi-stage chemical & pharmaceutical batch recipe 
 *              execution engine featuring 16-state sequential control,
 *              non-linear thermodynamics, adaptive dosing integration,
 *              tolerance checking matrices, multidimensional arrays,
 *              audit trails, methods, actions, and properties.
 *******************************************************************************)
{attribute 'reflection'}
{attribute 'no_explicit_call' := 'Run cyclic supervisor via instance call'}
FUNCTION_BLOCK FB_Sample_BatchRecipeExecutionEngine
VAR_INPUT
    bMasterEnable              : BOOL                := FALSE;                (* Master supervisor enable *)
    bStartBatchCommand         : BOOL                := FALSE;                (* Initiate new batch processing cycle *)
    bHoldBatchCommand          : BOOL                := FALSE;                (* Pause active processing stage *)
    bResumeBatchCommand        : BOOL                := FALSE;                (* Resume held processing stage *)
    bAbortBatchCommand         : BOOL                := FALSE;                (* Immediate emergency batch abort *)
    bAcknowledgeAlarms         : BOOL                := FALSE;                (* Alarm acknowledgment pulse *)
    bManualOverrideActive      : BOOL                := FALSE;                (* Manual override permit *)
    bSanitizationBypass        : BOOL                := FALSE;                (* Maintenance CIP bypass mode *)
    nSelectedRecipeId          : DINT                := 101;                  (* Target recipe identifier [100..999] *)
    nTargetBatchUnits          : UDINT               := 500;                  (* Target units to produce in current run *)
    nProductionPriorityLevel   : INT                 := 2;                    (* 1=Low, 2=Standard, 3=Urgent, 4=Critical *)
    fTargetVolume_L            : LREAL               := 2500.0;               (* Main reactor target liquid volume [L] *)
    fTargetTemperature_C       : LREAL               := 68.5;                 (* Target reaction temperature in [C] *)
    fAgitatorSetpoint_RPM      : REAL                := 320.0;                (* Active mixing speed setpoint [RPM] *)
    fPressureCeiling_Bar       : LREAL               := 4.2;                  (* Maximum reactor overpressure limit [Bar] *)
    fMinimumViscosityThreshold : REAL                := 0.85;                 (* Lowest fluid viscosity allowed *)
    tMaxDosingDuration         : TIME                := T#45S;                (* Maximum allowable dosing timeout *)
    tThermalHoldDuration       : TIME                := T#2M30S;              (* Reaction soak duration *)
    tSamplingInterval          : TIME                := T#200MS;              (* Telemetry acquisition tick *)
    tDegasDwellTime            : TIME                := T#15S;                (* De-aeration dwell duration *)
    sBatchSerialNumber         : STRING(80)          := 'BATCH-2026-CH-9941'; (* Serialized tracking code *)
    arrStageTolerances         : ARRAY[1..6] OF REAL := [0.01, 0.02, 0.05, 0.08, 0.10, 0.15];
END_VAR
VAR_OUTPUT
    bBatchInExecution         : BOOL;        (* TRUE when recipe sequence is progressing *)
    bBatchPausedInHold        : BOOL;        (* TRUE when batch is paused in safe hold *)
    bBatchSuccessfullyDone    : BOOL;        (* Set high on successful recipe cycle end *)
    bCriticalAlarmTripped     : BOOL;        (* High on active alarm / shutdown trip *)
    bReactorAgitatorInterlock : BOOL;        (* Safety interlock status for agitator motor *)
    bVesselVentingActive      : BOOL;        (* Relief valve opened status *)
    eCurrentBatchPhase        : INT;         (* 0=Idle, 10=PreCheck, 20=Dosing, 30=Agitation... *)
    nActiveStepNumber         : INT;         (* Internal sub-sequence execution step *)
    nCompletedBatchCount      : UDINT;       (* Lifetime completed batch counter *)
    fActualLiquidVolume_L     : LREAL;       (* Current measured liquid volume [L] *)
    fActualTemperature_C      : LREAL;       (* Current core reaction temperature [C] *)
    fActualPressure_Bar       : LREAL;       (* Measured internal headspace pressure [Bar] *)
    fActualAgitatorSpeed_RPM  : REAL;        (* Tachometer feedback from agitator shaft *)
    fReactionYieldPercent     : REAL;        (* Calculated chemical conversion yield % *)
    fProcessThermalDuty_kW    : LREAL;       (* Computed thermal heating/cooling power *)
    fEstimatedViscosity_cP    : REAL;        (* Dynamic viscosity estimator *)
    nSystemErrorCode          : UDINT;       (* 0=OK, 16#E101=Overpressure, 16#E102=ThermalRunaway *)
    sDetailedStatusMessage    : STRING(255); (* Operator readable diagnostic line *)
    tElapsedTimeInActiveStep  : TIME;        (* Step execution stopwatch *)
END_VAR
VAR_IN_OUT
    stDiagnostics : ST_Sample_DiagnosticsStruct; (* Shared plant diagnostic bus *)
END_VAR
VAR
    // --- 1. Subordinate Function Blocks and Timers ---
    _fbSubController        : FB_Sample_StateMachineController;
    _fbTelemetryRingBuffer  : FB_Sample_DataRingBuffer;
    _fbRTrigStart           : R_TRIG;
    _fbRTrigHold            : R_TRIG;
    _fbRTrigResume          : R_TRIG;
    _fbRTrigAbort           : R_TRIG;
    _fbRTrigAckAlarms       : R_TRIG;
    _fbTonStepWatchdog      : TON;
    _fbTonSamplingTicker    : TON;
    _fbTonThermalSoakTimer  : TON;
    _fbTonPurgeSafetyTimer  : TON;
    _fbTonDegasDwellTimer   : TON;
    _fbTonAgitatorRampTimer : TON;

    // --- 2. State Machine Engine Registers ---
    _nMasterState            : INT := 0; (* Master batch sequencer index *)
    _nPreviousState          : INT := 0; (* Prior state before hold / interrupt *)
    _nSubStateStep           : INT := 0; (* Secondary sub-state counter *)
    _nRetryCounter           : INT := 0; (* Retry attempt accumulator *)
    _nActiveRecipeIndex      : INT := 1; (* Recipe table row selector *)
    _bHoldLatchActive        : BOOL;     (* Hold condition latch *)
    _bEmergencyDumpActive    : BOOL;     (* Emergency dump valve trigger *)
    _bThermalRunawayDetected : BOOL;     (* Exotherm anomaly detected *)

    // --- 3. Thermodynamic and Kinematic Process Variables ---
    _fIntegratedMassFlow_kg   : LREAL;        (* Dosed material mass accumulator *)
    _fHeatExchangerDeltaT_K   : LREAL;        (* Jacket-to-core temperature difference *)
    _fThermalConductivity     : REAL := 0.58; (* Media thermal conductivity [W/mK] *)
    _fPID_IntegralAccum       : LREAL;        (* Internal thermal PID accumulator *)
    _fPID_DerivativePrevErr   : LREAL;        (* Previous cycle thermal error *)
    _fPeakObservedPressure    : LREAL := 0.0; (* Maximum recorded headspace pressure *)
    _fCumulativeThermalEnergy : LREAL := 0.0; (* Total Joules absorbed by batch *)

    // --- 4. Matrices, Lookups, and Recipe Buffers ---
    _arrRecipeMatrix         : ARRAY[1..4, 1..6] OF LREAL := [
        100.0, 25.0, 50.0, 1.0, 5.0, 0.01,
        250.0, 45.0, 120.0, 2.5, 10.0, 0.02,
        500.0, 68.5, 320.0, 4.2, 15.0, 0.05,
        1000.0, 85.0, 450.0, 6.0, 25.0, 0.08
    ];
    _arrDosingComponentFlows : ARRAY[1..5] OF LREAL := [12.5, 8.4, 3.2, 1.1, 0.5];
    _arrQualityVarianceLog   : ARRAY[1..8] OF REAL  := [0.0, 0.0, 0.0, 0.0, 0.0, 0.0, 0.0, 0.0];
    _arrRawTelemetryLog      : ARRAY[1..16] OF LREAL;
    _arrCalibrationOffsets   : ARRAY[1..4] OF LREAL := [0.0, 0.0, 0.0, 0.0];

    // --- 5. Internal Strings and Diagnostic Text ---
    _sActiveStepName   : STRING(80) := 'IDLE_STANDBY';
    _sRecipeTitle      : STRING(80) := 'DEFAULT_SYNTHESIS_RECIPE';
    _sAuditTrailLatest : STRING(255);
    _sOperatorNotes    : STRING(80) := 'NO_OPERATOR_OVERRIDE_ACTIVE';
END_VAR
VAR_TEMP
    _nTempLoopIdxA          : INT;
    _nTempLoopIdxB          : INT;
    _nTempArrayScan         : INT;
    _fTempMassSum           : LREAL;
    _fTempEnergyJoules      : LREAL;
    _fTempErrorDelta        : LREAL;
    _fTempCorrectionFactor  : REAL;
    _bTempConditionMet      : BOOL;
    _bTempSafetyInterlockOk : BOOL;
END_VAR
VAR CONSTANT
    cMaxAllowedPressure_Bar  : LREAL := 7.5;
    cMaxAllowedTemp_C        : LREAL := 115.0;
    cMinimumAgitationSpeed   : REAL  := 50.0;
    cSpecificHeatCapacity    : LREAL := 4186.0; (* Water equivalent J/(kg*K) *)
    cGravitationalAccel      : LREAL := 9.80665;
    cAtmosphericPressure_Bar : LREAL := 1.01325;
END_VAR

// =============================================================================
// 1. EVALUATE HARDWARE INPUT TRIGGERS & SAFETY INTERLOCKS
// =============================================================================
{region "Safety Interlock and Signal Ingestion"}
    _fbRTrigStart(CLK := bStartBatchCommand);
    _fbRTrigHold(CLK := bHoldBatchCommand);
    _fbRTrigResume(CLK := bResumeBatchCommand);
    _fbRTrigAbort(CLK := bAbortBatchCommand);
    _fbRTrigAckAlarms(CLK := bAcknowledgeAlarms);

    // Reset alarm latch on acknowledgment
    IF _fbRTrigAckAlarms.Q THEN
        bCriticalAlarmTripped  := FALSE;
        nSystemErrorCode       := 0;
        sDetailedStatusMessage := 'Alarms cleared by operator acknowledgment.';
END_IF

    // Emergency abort always forces state to safety shutdown
    IF _fbRTrigAbort.Q OR (bMasterEnable = FALSE AND _nMasterState > 0) THEN
        _nMasterState       := 900; // Emergency Shutdown & Depressurize
        _bEmergencyDumpActive  := TRUE;
        sDetailedStatusMessage := 'EMERGENCY ABORT TRIGGERED - Depressurizing reactor.';
END_IF

    // Cyclic Step Watchdog Timer
    _fbTonStepWatchdog(IN := (_nMasterState > 0 AND _nMasterState < 800), PT := tMaxDosingDuration);

    IF _fbTonStepWatchdog.Q AND NOT bCriticalAlarmTripped THEN
        bCriticalAlarmTripped := TRUE;
        nSystemErrorCode      := 16#E001; // Step timeout fault
        sDetailedStatusMessage := 'CRITICAL FAULT: Active process step exceeded maximum watchdog duration.';
        _nMasterState         := 800;     // Fault Hold
END_IF

    // Cyclic Telemetry Sampler Ticker
    _fbTonSamplingTicker(IN := NOT _fbTonSamplingTicker.Q, PT := tSamplingInterval);

    IF _fbTonSamplingTicker.Q AND bMasterEnable THEN
        _fbTelemetryRingBuffer.M_Push(fValue := fActualTemperature_C);
        A_UpdateSensorAggregations();
END_IF

    // Track peak pressure observed during batch
    IF fActualPressure_Bar > _fPeakObservedPressure THEN
        _fPeakObservedPressure := fActualPressure_Bar;
END_IF

    // Safety interlock check for agitator motor
    A_CheckSafetyInterlocks();
{endregion}

// =============================================================================
// 2. MASTER RECIPE EXECUTION SEQUENCER (16-STATE ENGINE)
// =============================================================================
CASE _nMasterState OF

    0:
        // STATE 0: IDLE STANDBY
        _sActiveStepName         := 'IDLE_STANDBY';
        bBatchInExecution        := FALSE;
        bBatchPausedInHold       := FALSE;
        bBatchSuccessfullyDone   := FALSE;
        _bHoldLatchActive        := FALSE;
        _bThermalRunawayDetected := FALSE;
        _nSubStateStep           := 0;
        _nRetryCounter           := 0;
        fActualAgitatorSpeed_RPM := 0.0;
        fProcessThermalDuty_kW   := 0.0;

        IF _fbRTrigStart.Q AND bMasterEnable AND NOT bCriticalAlarmTripped THEN
            IF nSelectedRecipeId >= 100 AND_THEN nSelectedRecipeId <= 999 THEN
                _bTempSafetyInterlockOk := TRUE;
                A_PerformSanityDiagnostics();

                IF _bTempSafetyInterlockOk THEN
                    _nMasterState     := 10; // Proceed to Recipe Ingestion & PreCheck
                    bBatchInExecution      := TRUE;
                    sDetailedStatusMessage := 'Batch cycle initiated. Verifying recipe parameters...';
                ELSE
                    nSystemErrorCode       := 16#E010;
                    sDetailedStatusMessage := 'Cannot start batch: Pre-startup safety diagnostics failed.';
                END_IF
            ELSE
                nSystemErrorCode       := 16#E011;
                sDetailedStatusMessage := 'Cannot start batch: Invalid Recipe ID provided.';
            END_IF
        END_IF

    10:
        // STATE 10: RECIPE INGESTION & MATRIX LOOKUP
        _sActiveStepName := 'RECIPE_INGESTION_AND_PRECHECK';
        _nSubStateStep   := 1;

        _bTempConditionMet := M_LoadRecipeParameters(nRecipeId := nSelectedRecipeId);

        IF _bTempConditionMet THEN
            _fIntegratedMassFlow_kg   := 0.0;
            _fPID_IntegralAccum       := 0.0;
            _fPID_DerivativePrevErr   := 0.0;
            _fCumulativeThermalEnergy := 0.0;
            _fPeakObservedPressure    := cAtmosphericPressure_Bar;
            fActualLiquidVolume_L   := 50.0; // Residual tare volume
            fActualTemperature_C    := 22.0; // Ambient starting temp
            fActualPressure_Bar := cAtmosphericPressure_Bar;
            _nMasterState           := 20;   // Advance to Inert Gas Purging
            sDetailedStatusMessage  := 'Recipe loaded successfully. Initiating nitrogen purge.';
        ELSE
            nSystemErrorCode       := 16#E020;
            sDetailedStatusMessage := 'Recipe loading failed: Incompatible parameter constraints.';
            _nMasterState    := 800; // Fault state
        END_IF

    20:
        // STATE 20: INERT GAS PURGE & OXYGEN DISPLACEMENT
        _sActiveStepName := 'NITROGEN_INERT_PURGE';
        _nSubStateStep   := 2;

        _fbTonPurgeSafetyTimer(IN := TRUE, PT := T#3S);

        IF _fbTonPurgeSafetyTimer.Q THEN
            _fbTonPurgeSafetyTimer(IN := FALSE);
            _nMasterState          := 30; // Advance to Liquid Pre-Dosing
            sDetailedStatusMessage := 'Purge cycle complete. Commencing raw material dosing.';
        END_IF

    30:
        // STATE 30: RAW MATERIAL LIQUID DOSING
        _sActiveStepName := 'RAW_MATERIAL_DOSING';
        _nSubStateStep   := 3;

        // Check for hold request
        IF _fbRTrigHold.Q THEN
            _nPreviousState := 30;
            _nMasterState   := 700; // Pause in safe hold
        ELSE
            _bTempConditionMet := M_ExecuteDosingSequence(fTargetVol := fTargetVolume_L, fCurrentVol := fActualLiquidVolume_L, arrFlowRates := _arrDosingComponentFlows);

            IF _bTempConditionMet THEN
                _nMasterState          := 35; // Advance to De-Aeration Dwell
                sDetailedStatusMessage := 'Dosing complete. Commencing de-aeration dwell.';
            ELSIF fActualPressure_Bar > fPressureCeiling_Bar THEN
                nSystemErrorCode       := 16#E030;
                sDetailedStatusMessage := 'Overpressure condition detected during liquid dosing!';
                _nMasterState          := 800;
            END_IF
        END_IF

    35:
        // STATE 35: DE-AERATION & HEADSPACE STABILIZATION
        _sActiveStepName := 'DE_AERATION_HEADSPACE_DWELL';
        _nSubStateStep   := 4;

        _fbTonDegasDwellTimer(IN := TRUE, PT := tDegasDwellTime);

        IF _fbTonDegasDwellTimer.Q THEN
            _fbTonDegasDwellTimer(IN := FALSE);
            _nMasterState          := 40; // Advance to Agitation Ramp
            sDetailedStatusMessage := 'De-aeration complete. Commencing agitator speed ramp.';
        END_IF

    40:
        // STATE 40: AGITATION ACCELERATION & VISCOSITY ADAPTATION
        _sActiveStepName := 'AGITATION_SPEED_RAMP';
        _nSubStateStep   := 5;

        IF fActualAgitatorSpeed_RPM < fAgitatorSetpoint_RPM THEN
            fActualAgitatorSpeed_RPM := fActualAgitatorSpeed_RPM + 15.0;

            IF fActualAgitatorSpeed_RPM > fAgitatorSetpoint_RPM THEN
                fActualAgitatorSpeed_RPM := fAgitatorSetpoint_RPM;
            END_IF
        END_IF

        fEstimatedViscosity_cP := M_CalculateDynamicViscosity(fTemperature := fActualTemperature_C, fAgitationRPM := fActualAgitatorSpeed_RPM);

        IF fActualAgitatorSpeed_RPM >= fAgitatorSetpoint_RPM THEN
            _nMasterState          := 50; // Advance to Thermal Ramp & Reaction
            sDetailedStatusMessage := 'Agitator at target speed. Engaging heating jacket.';
        END_IF

    50:
        // STATE 50: THERMAL HEATING RAMP & TEMPERATURE SOAK
        _sActiveStepName := 'THERMAL_HEATING_RAMP';
        _nSubStateStep   := 6;

        M_RegulateThermalEquilibrium(fTargetTemp := fTargetTemperature_C, fCoreTemp := fActualTemperature_C, fJacketDeltaT := _fHeatExchangerDeltaT_K, fDutyOutput => fProcessThermalDuty_kW);

        // Check if temperature reached thermal equilibrium band
        IF ABS(fActualTemperature_C - fTargetTemperature_C) <= 0.75 THEN
            _fbTonThermalSoakTimer(IN := TRUE, PT := tThermalHoldDuration);
            sDetailedStatusMessage := 'Thermal equilibrium reached. Maintaining reaction soak.';

            IF _fbTonThermalSoakTimer.Q THEN
                _fbTonThermalSoakTimer(IN := FALSE);
                _nMasterState          := 60; // Advance to Quality Gate Evaluation
                sDetailedStatusMessage := 'Reaction soak completed. Evaluating quality metrics.';
            END_IF
        ELSE
            _fbTonThermalSoakTimer(IN := FALSE);
        END_IF

    60:
        // STATE 60: QUALITY ASSURANCE & SPECTRAL DENSITY EVALUATION
        _sActiveStepName := 'QUALITY_ASSURANCE_GATE';
        _nSubStateStep   := 7;

        _bTempConditionMet := M_MonitorQualityAssuranceGate(arrTolerances := arrStageTolerances, fYieldPercent => fReactionYieldPercent);

        IF _bTempConditionMet AND fReactionYieldPercent >= 92.5 THEN
            _nMasterState          := 70; // Advance to Product Cooling & Quench
            sDetailedStatusMessage := 'Quality gate passed. Beginning controlled cooling quench.';
        ELSE
            IF _nRetryCounter < 2 THEN
                _nRetryCounter := _nRetryCounter + 1;
                _nMasterState  := 50; // Re-enter thermal soak to complete conversion
                sDetailedStatusMessage := 'Quality gate borderline. Extending thermal conversion.';
            ELSE
                nSystemErrorCode       := 16#E060;
                sDetailedStatusMessage := 'Quality gate failed: Yield below minimum threshold.';
                _nMasterState    := 800; // Fault hold
            END_IF
        END_IF

    70:
        // STATE 70: PRODUCT COOLING & THERMAL QUENCH
        _sActiveStepName := 'CONTROLLED_PRODUCT_COOLING';
        _nSubStateStep   := 8;

        IF fActualTemperature_C > 30.0 THEN
            fActualTemperature_C   := fActualTemperature_C - 2.5;
            fProcessThermalDuty_kW := -35.0; // Active chilled cooling
        ELSE
            fProcessThermalDuty_kW := 0.0;
            _nMasterState          := 80; // Advance to Discharge Sequence
            sDetailedStatusMessage := 'Cooling complete. Ready for product discharge.';
        END_IF

    80:
        // STATE 80: PRODUCT DISCHARGE SEQUENCE
        _sActiveStepName := 'PRODUCT_DISCHARGE';
        _nSubStateStep   := 9;

        IF fActualLiquidVolume_L > 10.0 THEN
            fActualLiquidVolume_L := fActualLiquidVolume_L - 85.0;

            IF fActualLiquidVolume_L < 10.0 THEN
                fActualLiquidVolume_L := 10.0;
            END_IF
        ELSE
            IF bSanitizationBypass THEN
                _nMasterState          := 100; // Skip CIP, jump to Completion
                sDetailedStatusMessage := 'CIP bypass enabled. Finalizing batch audit log.';
            ELSE
                _nMasterState          := 90; // Advance to Clean-In-Place (CIP)
                sDetailedStatusMessage := 'Discharge complete. Commencing CIP sanitation cycle.';
            END_IF
        END_IF

    90:
        // STATE 90: CLEAN-IN-PLACE (CIP) SANITATION SEQUENCE
        _sActiveStepName := 'CLEAN_IN_PLACE_CIP';
        _nSubStateStep   := 10;

        // Sub-controller execution for wash sequence
        _fbSubController(bStart := TRUE, bStop := FALSE, bReset := FALSE, tStepTimeout := T#4S);

        IF _fbSubController.eCurrentState = 90 THEN
            _fbSubController(bStart := FALSE, bStop := TRUE, bReset := TRUE);
            _nMasterState          := 100; // Batch Completion
            sDetailedStatusMessage := 'CIP cycle finished. Finalizing batch audit log.';
        END_IF

    100:
        // STATE 100: BATCH COMPLETION & AUDIT GENERATION
        _sActiveStepName       := 'BATCH_COMPLETED_SUCCESS';
        bBatchInExecution      := FALSE;
        bBatchSuccessfullyDone := TRUE;
        nCompletedBatchCount   := nCompletedBatchCount + 1;

        M_GenerateAuditTrailSummary(sSerial := sBatchSerialNumber);
        A_CalculateEnergyConsumption();

        sDetailedStatusMessage := 'Batch process successfully finished with full audit compliance.';
        _nMasterState          := 0; // Return to Standby

    700:
        // STATE 700: PAUSED IN SAFE HOLD
        _sActiveStepName       := 'PAUSED_SAFE_HOLD';
        bBatchPausedInHold     := TRUE;
        bBatchInExecution      := FALSE;
        fProcessThermalDuty_kW := 0.0;

        IF _fbRTrigResume.Q AND NOT bCriticalAlarmTripped THEN
            bBatchPausedInHold     := FALSE;
            bBatchInExecution      := TRUE;
            _nMasterState          := _nPreviousState;
            sDetailedStatusMessage := 'Process resumed from operator hold.';
        END_IF

    800:
        // STATE 800: FAULT STATE & ALARM TRIP
        _sActiveStepName         := 'FAULT_ALARM_HOLD';
        bCriticalAlarmTripped    := TRUE;
        bBatchInExecution        := FALSE;
        fProcessThermalDuty_kW   := 0.0;
        fActualAgitatorSpeed_RPM := 0.0;

        IF _fbRTrigAckAlarms.Q AND nSystemErrorCode = 0 THEN
            _nMasterState          := 0;
            sDetailedStatusMessage := 'Fault state reset. Engine returned to idle.';
        END_IF

    900:
        // STATE 900: EMERGENCY DEPRESSURIZE & DUMP
        _sActiveStepName := 'EMERGENCY_DEPRESSURIZE_DUMP';
        M_EmergencyDepressurizeAndDump();

        IF fActualPressure_Bar <= 1.05 AND fActualLiquidVolume_L <= 5.0 THEN
            _bEmergencyDumpActive  := FALSE;
            _nMasterState          := 800; // Transition to Fault state
            sDetailedStatusMessage := 'Emergency depressurization complete. Awaiting supervisor inspection.';
        END_IF

ELSE
    _nMasterState          := 800;
    nSystemErrorCode       := 16#E999;
    sDetailedStatusMessage := 'FATAL: Unknown state machine index encountered.';
END_CASE

eCurrentBatchPhase := _nMasterState;
nActiveStepNumber  := _nSubStateStep;

ACTION A_CalculateEnergyConsumption:
// Compute total thermal energy integrated over batch execution
_fTempEnergyJoules     := fActualLiquidVolume_L * cSpecificHeatCapacity * (fActualTemperature_C - 20.0);
fProcessThermalDuty_kW := _fTempEnergyJoules / (3600.0 * 1000.0);
END_ACTION

ACTION A_CheckSafetyInterlocks:
// Ensure agitator cannot run if vessel is empty or overpressurized
bReactorAgitatorInterlock := (fActualLiquidVolume_L >= 25.0) AND_THEN (fActualPressure_Bar <= fPressureCeiling_Bar) AND_THEN (NOT bCriticalAlarmTripped);

IF NOT bReactorAgitatorInterlock THEN
    fActualAgitatorSpeed_RPM := 0.0;
END_IF
END_ACTION

ACTION A_PerformSanityDiagnostics:
// Validate all physical sensors before allowing batch sequence launch
_bTempSafetyInterlockOk := (fActualPressure_Bar < cMaxAllowedPressure_Bar) AND_THEN (fActualTemperature_C < cMaxAllowedTemp_C) AND_THEN (NOT bCriticalAlarmTripped);
END_ACTION

ACTION A_UpdateSensorAggregations:
// Update plant diagnostics structure
stDiagnostics.nLightCount         := 4;
stDiagnostics.fArtificialLevelSum := TO_REAL(fActualLiquidVolume_L * 0.1);
stDiagnostics.fHumiditySensor     := TO_REAL(fActualTemperature_C * 0.5);
END_ACTION

METHOD M_CalculateDynamicViscosity : REAL
VAR_INPUT
    fTemperature  : LREAL;
    fAgitationRPM : REAL;
END_VAR
VAR
    _fBaseViscosity : REAL := 1.25;
    _fShearThinning : REAL;
END_VAR
_fShearThinning             := 1.0 / (1.0 + (fAgitationRPM * 0.002));
M_CalculateDynamicViscosity := _fBaseViscosity * _fShearThinning * TO_REAL(EXP(-0.015 * (fTemperature - 20.0)));
END_METHOD

METHOD M_CalibrateVesselSensors : BOOL
VAR_INPUT
    arrReferencePressures : ARRAY[1..4] OF LREAL;
    arrReferenceTemps     : ARRAY[1..4] OF LREAL;
END_VAR
VAR
    _nIndex : INT;
    _fDelta : LREAL;
END_VAR
FOR _nIndex := 1 TO 4 DO
    _fDelta                         := arrReferencePressures[_nIndex] - cAtmosphericPressure_Bar;
    _arrCalibrationOffsets[_nIndex] := _fDelta * 0.01;
END_FOR

M_CalibrateVesselSensors := TRUE;
END_METHOD

METHOD M_ComputeReactionKinetics : LREAL
VAR_INPUT
    fConcentrationA : LREAL;
    fConcentrationB : LREAL;
    fCoreTempK      : LREAL;
END_VAR
VAR
    _fActivationEnergy : LREAL := 45000.0; // J/mol
    _fGasConstant      : LREAL := 8.31446; // J/(mol*K)
    _fPreExpFactor     : LREAL := 1.25E6;
    _fRateConstant     : LREAL;
    _fReactionRate     : LREAL;
END_VAR
IF fCoreTempK <= 273.15 THEN
    M_ComputeReactionKinetics := 0.0;
    RETURN;
END_IF

// Arrhenius reaction rate constant approximation: k = A * exp(-Ea / (R * T))
_fRateConstant := _fPreExpFactor * EXP(-_fActivationEnergy / (_fGasConstant * fCoreTempK));

// Second-order rate law: r = k * [A] * [B]
_fReactionRate := _fRateConstant * fConcentrationA * fConcentrationB;

M_ComputeReactionKinetics := _fReactionRate;
END_METHOD

METHOD M_EmergencyDepressurizeAndDump : BOOL
VAR
    _fPressureDropRate : LREAL := 0.25;
    _fLiquidDumpRate   : LREAL := 150.0;
END_VAR
// Depressurize vessel towards atmospheric baseline
IF fActualPressure_Bar > cAtmosphericPressure_Bar THEN
    fActualPressure_Bar := fActualPressure_Bar - _fPressureDropRate;

    IF fActualPressure_Bar < cAtmosphericPressure_Bar THEN
        fActualPressure_Bar := cAtmosphericPressure_Bar;
    END_IF
END_IF

// Open emergency bottom dump valve to quench pit
IF fActualLiquidVolume_L > 0.0 THEN
    fActualLiquidVolume_L := fActualLiquidVolume_L - _fLiquidDumpRate;

    IF fActualLiquidVolume_L < 0.0 THEN
        fActualLiquidVolume_L := 0.0;
    END_IF
END_IF

// Stop all heating/cooling systems immediately
fProcessThermalDuty_kW   := 0.0;
fActualAgitatorSpeed_RPM := 0.0;

M_EmergencyDepressurizeAndDump := (fActualPressure_Bar <= cAtmosphericPressure_Bar AND fActualLiquidVolume_L <= 0.0);
END_METHOD

METHOD PUBLIC M_EstimateExothermicRunawayRisk : REAL
VAR_INPUT
    fReactionRate_mol_L_s  : LREAL;
    fCoolingCapacity_kW    : LREAL;
    fHeatOfReaction_kJ_mol : LREAL;
END_VAR
VAR
    _fHeatGeneration_kW : LREAL;
    _fRunawayRiskRatio  : LREAL;
END_VAR
// Calculate instantaneous heat generation rate
_fHeatGeneration_kW := fReactionRate_mol_L_s * fHeatOfReaction_kJ_mol * fActualLiquidVolume_L;

IF fCoolingCapacity_kW > 0.001 THEN
    _fRunawayRiskRatio := _fHeatGeneration_kW / fCoolingCapacity_kW;
ELSE
    _fRunawayRiskRatio := 10.0;
END_IF

IF _fRunawayRiskRatio > 1.0 THEN
    bCriticalAlarmTripped  := TRUE;
    sDetailedStatusMessage := 'THERMAL RUNAWAY RISK: Heat generation exceeds cooling capacity!';
END_IF

M_EstimateExothermicRunawayRisk := TO_REAL(_fRunawayRiskRatio);
END_METHOD

METHOD M_ExecuteDosingSequence : BOOL
VAR_INPUT
    fTargetVol   : LREAL;
    fCurrentVol  : LREAL;
    arrFlowRates : ARRAY[1..5] OF LREAL;
END_VAR
VAR
    _nCompIdx   : INT;
    _fTotalFlow : LREAL := 0.0;
    _fIncrement : LREAL;
END_VAR
IF fTargetVol <= 0.0 THEN
    M_ExecuteDosingSequence := FALSE;
    RETURN;
END_IF

// Aggregate flow rate contributions across all 5 dosing pumps
FOR _nCompIdx := 1 TO 5 DO
    IF arrFlowRates[_nCompIdx] > 0.0 THEN
        _fTotalFlow := _fTotalFlow + arrFlowRates[_nCompIdx];
    END_IF
END_FOR

// Scale step volume increment based on aggregate flow rate
_fIncrement             := (_fTotalFlow * 0.25) / 60.0;
fActualLiquidVolume_L   := fActualLiquidVolume_L + _fIncrement;
_fIntegratedMassFlow_kg := _fIntegratedMassFlow_kg + (_fIncrement * 1.025);

// Update vessel headspace pressure pneumatics
fActualPressure_Bar := cAtmosphericPressure_Bar + ((fActualLiquidVolume_L / fTargetVol) * 1.85);

// Check if vessel dosing is complete
IF fActualLiquidVolume_L >= fTargetVol THEN
    fActualLiquidVolume_L   := fTargetVol;
    M_ExecuteDosingSequence := TRUE;
ELSE
    M_ExecuteDosingSequence := FALSE;
END_IF
END_METHOD

METHOD M_FormatBatchReportPayload : STRING(255)
VAR_INPUT
    sBatchTag : STRING(50);
END_VAR
VAR
    _sResult : STRING(255);
    _sVolume : STRING(30);
    _sYield  : STRING(30);
    _sPress  : STRING(30);
END_VAR
_sVolume := LREAL_TO_STRING(fActualLiquidVolume_L);
_sYield  := REAL_TO_STRING(fReactionYieldPercent);
_sPress  := LREAL_TO_STRING(fActualPressure_Bar);

_sResult := CONCAT('{"batch_id":"', sBatchTag);
_sResult := CONCAT(_sResult, '","volume_l":');
_sResult := CONCAT(_sResult, _sVolume);
_sResult := CONCAT(_sResult, ',"yield_pct":');
_sResult := CONCAT(_sResult, _sYield);
_sResult := CONCAT(_sResult, ',"pressure_bar":');
_sResult := CONCAT(_sResult, _sPress);
_sResult := CONCAT(_sResult, ',"status":"COMPLETE"}');

M_FormatBatchReportPayload := _sResult;
END_METHOD

METHOD M_GenerateAuditTrailSummary : BOOL
VAR_INPUT
    sSerial : STRING(80);
END_VAR
VAR
    _sBatchCode : STRING(80);
    _sYieldText : STRING(30);
    _sTempText  : STRING(30);
END_VAR
_sBatchCode := sSerial;
_sYieldText := REAL_TO_STRING(fReactionYieldPercent);
_sTempText  := LREAL_TO_STRING(fActualTemperature_C);

_sAuditTrailLatest := CONCAT('BATCH COMPLIANCE AUDIT | ID: ', _sBatchCode);
_sAuditTrailLatest := CONCAT(_sAuditTrailLatest, ' | Yield: ');
_sAuditTrailLatest := CONCAT(_sAuditTrailLatest, _sYieldText);
_sAuditTrailLatest := CONCAT(_sAuditTrailLatest, '% | Final Temp: ');
_sAuditTrailLatest := CONCAT(_sAuditTrailLatest, _sTempText);
_sAuditTrailLatest := CONCAT(_sAuditTrailLatest, ' C | Status: VALIDATED_PASSED');

sDetailedStatusMessage      := _sAuditTrailLatest;
M_GenerateAuditTrailSummary := TRUE;
END_METHOD

METHOD M_LoadRecipeParameters : BOOL
VAR_INPUT
    nRecipeId : DINT;
END_VAR
VAR
    _nRowIndex    : INT;
    _nColIndex    : INT;
    _fTargetMass  : LREAL;
    _fDensityCorr : REAL;
END_VAR
IF nRecipeId < 100 OR nRecipeId > 999 THEN
    M_LoadRecipeParameters := FALSE;
    RETURN;
END_IF

// Multi-tier recipe row selection based on recipe identifier
IF nRecipeId >= 100 AND nRecipeId < 200 THEN
    _nRowIndex    := 1;
    _sRecipeTitle := 'STANDARD_ORGANIC_SYNTHESIS';
ELSIF nRecipeId >= 200 AND nRecipeId < 400 THEN
    _nRowIndex    := 2;
    _sRecipeTitle := 'HIGH_VISCOSITY_POLYMERIC_BLEND';
ELSIF nRecipeId >= 400 AND nRecipeId < 700 THEN
    _nRowIndex    := 3;
    _sRecipeTitle := 'EXOTHERMIC_CATALYTIC_REACTION';
ELSE
    _nRowIndex    := 4;
    _sRecipeTitle := 'SPECIALTY_PHARMACEUTICAL_BATCH';
END_IF

_nActiveRecipeIndex := _nRowIndex;

// Extract recipe parameters from internal recipe matrix
fTargetVolume_L       := _arrRecipeMatrix[_nRowIndex, 1];
fTargetTemperature_C  := _arrRecipeMatrix[_nRowIndex, 2];
fAgitatorSetpoint_RPM := TO_REAL(_arrRecipeMatrix[_nRowIndex, 3]);
fPressureCeiling_Bar  := _arrRecipeMatrix[_nRowIndex, 4];

// Validate thermodynamic sanity
IF fTargetTemperature_C > cMaxAllowedTemp_C OR_ELSE fPressureCeiling_Bar > cMaxAllowedPressure_Bar THEN
    M_LoadRecipeParameters := FALSE;
    RETURN;
END_IF

// Calculate predicted mass from volume and thermal expansion curve
_fDensityCorr := 1.0 - (TO_REAL(fTargetTemperature_C - 20.0) * 0.00045);
_fTargetMass  := fTargetVolume_L * TO_LREAL(_fDensityCorr);

M_LoadRecipeParameters := TRUE;
END_METHOD

METHOD M_MonitorQualityAssuranceGate : BOOL
VAR_INPUT
    arrTolerances : ARRAY[1..6] OF REAL;
END_VAR
VAR_OUTPUT
    fYieldPercent : REAL;
END_VAR
VAR
    _nIdx          : INT;
    _fVarianceSum  : REAL := 0.0;
    _fMeanVar      : REAL;
    _bAllWithinTol : BOOL := TRUE;
END_VAR
// Iterate over tolerance metrics
FOR _nIdx := 1 TO 6 DO
    _arrQualityVarianceLog[_nIdx] := TO_REAL(ABS(fActualTemperature_C - fTargetTemperature_C) / fTargetTemperature_C);
    _fVarianceSum                 := _fVarianceSum + _arrQualityVarianceLog[_nIdx];

    IF _arrQualityVarianceLog[_nIdx] > arrTolerances[_nIdx] THEN
        _bAllWithinTol := FALSE;
    END_IF
END_FOR

_fMeanVar := _fVarianceSum / 6.0;

// Derive chemical synthesis yield percentage from variance metrics
IF _bAllWithinTol THEN
    fYieldPercent := 98.5 - (_fMeanVar * 100.0);

    IF fYieldPercent > 99.8 THEN
        fYieldPercent := 99.8;
    END_IF

    M_MonitorQualityAssuranceGate := TRUE;
ELSE
    fYieldPercent                 := 88.0 - (_fMeanVar * 120.0);
    M_MonitorQualityAssuranceGate := FALSE;
END_IF
END_METHOD

METHOD M_RegulateThermalEquilibrium : BOOL
VAR_INPUT
    fTargetTemp   : LREAL;
    fCoreTemp     : LREAL;
    fJacketDeltaT : LREAL;
END_VAR
VAR_OUTPUT
    fDutyOutput : LREAL;
END_VAR
VAR
    _fKp          : LREAL := 4.5;
    _fKi          : LREAL := 0.08;
    _fKd          : LREAL := 1.2;
    _fError       : LREAL;
    _fP_Term      : LREAL;
    _fI_Term      : LREAL;
    _fD_Term      : LREAL;
    _fTotalOutput : LREAL;
END_VAR
_fError := fTargetTemp - fCoreTemp;

// Proportional Term
_fP_Term := _fKp * _fError;

// Integral Term with Anti-Windup Clamping
_fPID_IntegralAccum := _fPID_IntegralAccum + (_fError * 0.1);

IF _fPID_IntegralAccum > 500.0 THEN
    _fPID_IntegralAccum := 500.0;
ELSIF _fPID_IntegralAccum < -500.0 THEN
    _fPID_IntegralAccum := -500.0;
END_IF

_fI_Term := _fKi * _fPID_IntegralAccum;

// Derivative Term
_fD_Term                := _fKd * (_fError - _fPID_DerivativePrevErr);
_fPID_DerivativePrevErr := _fError;

// Combined PID Thermal Duty
_fTotalOutput := _fP_Term + _fI_Term + _fD_Term;

// Clamp Thermal Output to [-100.0 kW Chilling .. +100.0 kW Heating]
IF _fTotalOutput > 100.0 THEN
    fDutyOutput := 100.0;
ELSIF _fTotalOutput < -100.0 THEN
    fDutyOutput := -100.0;
ELSE
    fDutyOutput := _fTotalOutput;
END_IF

// Simulate thermodynamic heat transfer response on core temperature
IF fDutyOutput > 0.0 THEN
    fActualTemperature_C := fActualTemperature_C + (fDutyOutput * 0.012);
ELSE
    fActualTemperature_C := fActualTemperature_C + (fDutyOutput * 0.018);
END_IF

M_RegulateThermalEquilibrium := (ABS(_fError) < 0.5);
END_METHOD

METHOD M_ValidateQualityAssuranceMatrix : BOOL
VAR_INPUT
    arrReferenceMatrix : ARRAY[1..4, 1..6] OF LREAL;
    fTightTolerance    : LREAL;
END_VAR
VAR
    _nRow    : INT;
    _nCol    : INT;
    _fDelta  : LREAL;
    _bPassed : BOOL := TRUE;
END_VAR
FOR _nRow := 1 TO 4 DO
    FOR _nCol := 1 TO 6 DO
        _fDelta := ABS(_arrRecipeMatrix[_nRow, _nCol] - arrReferenceMatrix[_nRow, _nCol]);

        IF _fDelta > fTightTolerance THEN
            _bPassed := FALSE;
            EXIT;
        END_IF
    END_FOR
    IF NOT _bPassed THEN
        EXIT;
    END_IF
END_FOR

M_ValidateQualityAssuranceMatrix := _bPassed;
END_METHOD

PROPERTY P_ActiveRecipeName : STRING(80)
GET
P_ActiveRecipeName := _sRecipeTitle;
END_GET
SET
_sRecipeTitle := P_ActiveRecipeName;
END_SET
END_PROPERTY

PROPERTY P_DosingAccuracyPct : REAL
GET
VAR
    _fDev : LREAL;
END_VAR
IF fTargetVolume_L > 0.0 THEN
    _fDev               := ABS(fActualLiquidVolume_L - fTargetVolume_L) / fTargetVolume_L;
    P_DosingAccuracyPct := TO_REAL((1.0 - _fDev) * 100.0);
ELSE
    P_DosingAccuracyPct := 100.0;
END_IF
END_GET
END_PROPERTY

PROPERTY P_OverallBatchProgress : REAL
GET
IF _nMasterState = 0 THEN
    P_OverallBatchProgress := 0.0;
ELSIF _nMasterState >= 100 THEN
    P_OverallBatchProgress := 100.0;
ELSE
    P_OverallBatchProgress := (TO_REAL(_nMasterState) / 100.0) * 100.0;
END_IF
END_GET
END_PROPERTY

PROPERTY P_ReactorThermodynamicHealth : REAL
GET
VAR
    _fHealthIndex : REAL := 100.0;
END_VAR
IF fActualPressure_Bar > (fPressureCeiling_Bar * 0.9) THEN
    _fHealthIndex := _fHealthIndex - 35.0;
END_IF

IF fActualTemperature_C > (cMaxAllowedTemp_C * 0.85) THEN
    _fHealthIndex := _fHealthIndex - 40.0;
END_IF

IF _fHealthIndex < 0.0 THEN
    _fHealthIndex := 0.0;
END_IF

P_ReactorThermodynamicHealth := _fHealthIndex;
END_GET
END_PROPERTY

END_FUNCTION_BLOCK

// ---- samples/FB_Sample_HighDensityDataAnalyticsLogger.TcPOU
(*******************************************************************************
 * POU Name:    FB_Sample_HighDensityDataAnalyticsLogger
 * Description: High-density industrial telemetry data logger, online statistical
 *              moment analyzer (Welford algorithm, skewness, kurtosis),
 *              CUSUM drift anomaly detector, Delta-RLE data compression engine,
 *              CRC32 checksum framing, 1D Kalman filtering, InfluxDB formatters,
 *              methods, actions, and properties (>1000 lines).
 *******************************************************************************)
{attribute 'reflection'}
{attribute 'no_explicit_call' := 'Run cyclic analytics logger via instance call'}
FUNCTION_BLOCK FB_Sample_HighDensityDataAnalyticsLogger
VAR_INPUT
    bLoggerMasterEnable      : BOOL                  := FALSE;       (* Master telemetry acquisition permit *)
    bTriggerSnapshotLog      : BOOL                  := FALSE;       (* Force immediate data frame capture *)
    bClearBufferCommand      : BOOL                  := FALSE;       (* Purge internal memory ring buffer *)
    bForceFlushToSink        : BOOL                  := FALSE;       (* Trigger writeout to persistent sink *)
    bAcknowledgeAnomalyAlarm : BOOL                  := FALSE;       (* Operator anomaly alarm acknowledgment *)
    bEnableRLECompression    : BOOL                  := TRUE;        (* Activate Delta-RLE payload compression *)
    bEnableKalmanFiltering   : BOOL                  := TRUE;        (* In-line 1D Kalman filter enable *)
    nSamplingFrequency_Hz    : UDINT                 := 500;         (* Telemetry sample rate [Hz] *)
    nActiveChannelBitmask    : DWORD                 := 16#FFFFFFFF; (* 32-channel active channel selection mask *)
    nArchivePartitionId      : DINT                  := 101;         (* Target storage partition number *)
    fZScoreAlarmThreshold    : LREAL                 := 3.25;        (* Anomaly trigger statistical sigma limit *)
    fCusumSlackParameter     : LREAL                 := 0.5;         (* CUSUM reference slack constant k *)
    fCusumDecisionInterval   : LREAL                 := 4.5;         (* CUSUM alarm threshold parameter h *)
    fKalmanProcessNoise_Q    : LREAL                 := 0.01;        (* Process noise covariance Q *)
    fKalmanMeasureNoise_R    : LREAL                 := 0.1;         (* Measurement noise covariance R *)
    tMaxFlushTimeout         : TIME                  := T#5S;        (* Storage sink handshake timeout *)
    tHeartbeatInterval       : TIME                  := T#1S;        (* Periodic logger health tick *)
    sSinkEndpointURI         : STRING(80)            := 'https://telemetry.edge.internal:8443/v1/ingest';
    arrChannelScalingGains   : ARRAY[1..16] OF LREAL := [1.0, 1.0, 1.0, 1.0, 2.5, 2.5, 0.1, 0.1, 10.0, 10.0, 0.05, 0.05, 1.0, 1.0, 1.0, 1.0];
END_VAR
VAR_OUTPUT
    bLoggerActive            : BOOL;        (* High when telemetry engine is recording *)
    bBufferHalfFullWarning   : BOOL;        (* Buffer fill level > 50% *)
    bBufferOverflowFault     : BOOL;        (* Ring buffer saturated *)
    bProcessAnomalyDetected  : BOOL;        (* Critical statistical outlier tripped *)
    bSinkFlushInProgress     : BOOL;        (* Asynchronous disk/network write active *)
    bPayloadCompressed       : BOOL;        (* Compression pass successfully applied *)
    eCurrentLoggerPhase      : INT;         (* 0=Idle, 10=Sample, 20=Filter, 30=Welford... *)
    nTotalSamplesLogged      : ULINT;       (* Cumulative samples acquired *)
    nSamplesInCurrentFrame   : UDINT;       (* Samples packed into active frame *)
    nActiveAnomalyCount      : UDINT;       (* Cumulative outlier events detected *)
    nActivePartitionIndex    : DINT;        (* Active storage partition *)
    fBufferUtilizationPct    : REAL;        (* Ring buffer fill level [0..100%] *)
    fEffectiveDataThroughput : REAL;        (* Ingestion throughput in [kB/s] *)
    fOverallCompressionRatio : REAL;        (* Raw-to-compressed size ratio *)
    nComputedCRC32           : DWORD;       (* Frame integrity checksum *)
    nLoggerErrorCode         : UDINT;       (* 0=OK, 16#A001=Overflow, 16#A002=SinkTimeout *)
    sDetailedLoggerStatus    : STRING(255); (* Operator readable diagnostic line *)
    tElapsedTimeInActiveTick : TIME;        (* Step execution stopwatch *)
END_VAR
VAR_IN_OUT
    stDiagnostics : ST_Sample_DiagnosticsStruct; (* Shared plant diagnostic bus *)
END_VAR
VAR
    // --- 1. Subordinate Function Blocks and Timers ---
    _fbSinkStateController   : FB_Sample_StateMachineController;
    _fbRollingBufferPrimary  : FB_Sample_DataRingBuffer;
    _fbRTrigCapture          : R_TRIG;
    _fbRTrigClear            : R_TRIG;
    _fbRTrigFlush            : R_TRIG;
    _fbRTrigAckAnomaly       : R_TRIG;
    _fbTonFlushWatchdog      : TON;
    _fbTonHeartbeatTicker    : TON;
    _fbTonAcquisitionTicker  : TON;
    _fbTonAnomalySettleTimer : TON;

    // --- 2. State Machine Engine Registers ---
    _nMasterLoggerState      : INT   := 0;     (* Master logger sequence index *)
    _nPreviousLoggerState    : INT   := 0;     (* Previous state prior to pause *)
    _nFrameSequenceNumber    : UDINT := 0;     (* Frame counter for packet header *)
    _nRetryFlushAttempts     : INT   := 0;     (* Disk write retry count *)
    _bSinkHandshakeReady     : BOOL  := FALSE; (* External storage sink permit *)
    _bCusumDriftAlarmLatched : BOOL  := FALSE; (* Latched process drift alert *)

    // --- 3. Statistical Analysis Registers (Welford, Skewness & CUSUM) ---
    _arrChannelMean        : ARRAY[1..16] OF LREAL; (* Running sample mean *)
    _arrChannelM2_Accum    : ARRAY[1..16] OF LREAL; (* Second central moment accumulator *)
    _arrChannelM3_Accum    : ARRAY[1..16] OF LREAL; (* Third central moment accumulator *)
    _arrChannelM4_Accum    : ARRAY[1..16] OF LREAL; (* Fourth central moment accumulator *)
    _arrChannelVariance    : ARRAY[1..16] OF LREAL; (* Sample variance *)
    _arrChannelStdDev      : ARRAY[1..16] OF LREAL; (* Sample standard deviation *)
    _arrChannelSkewness    : ARRAY[1..16] OF LREAL; (* Sample skewness coefficient *)
    _arrChannelKurtosis    : ARRAY[1..16] OF LREAL; (* Sample kurtosis coefficient *)
    _arrChannelCusumPos    : ARRAY[1..16] OF LREAL; (* Positive CUSUM cumulative sum *)
    _arrChannelCusumNeg    : ARRAY[1..16] OF LREAL; (* Negative CUSUM cumulative sum *)
    _arrChannelRawReadings : ARRAY[1..16] OF LREAL; (* Instantaneous sensor ADC values *)
    _arrChannelFiltered    : ARRAY[1..16] OF LREAL; (* Low-pass filtered sensor stream *)
    _arrKalmanEstimate     : ARRAY[1..16] OF LREAL; (* 1D Kalman state estimate *)
    _arrKalmanCovariance   : ARRAY[1..16] OF LREAL := [1.0, 1.0, 1.0, 1.0, 1.0, 1.0, 1.0, 1.0, 1.0, 1.0, 1.0, 1.0, 1.0, 1.0, 1.0, 1.0];

    // --- 4. Frame Buffers, Checksums, and Lookups ---
    _arrRawFramePayloadWords : ARRAY[1..32] OF WORD;
    _arrCompressedFrameBytes : ARRAY[1..64] OF BYTE;
    _arrCRC32LookupTable     : ARRAY[0..15] OF DWORD;

    // --- 5. Internal Strings and Diagnostic Text ---
    _sActiveLoggerPhaseName  : STRING(80) := 'STANDBY_IDLE';
    _sPartitionDirectoryPath : STRING(80) := '/var/log/telemetry/partition_101/';
    _sLatestTelemetryJSON    : STRING(255);
    _sInfluxLineBuffer       : STRING(255);
END_VAR
VAR_TEMP
    _nTempChanIdx        : INT;
    _nTempByteScan       : INT;
    _fTempDeltaWelford   : LREAL;
    _fTempZScore         : LREAL;
    _fTempThroughputCalc : REAL;
    _bTempAnomalyInScan  : BOOL;
    _bTempFlushSuccess   : BOOL;
END_VAR
VAR CONSTANT
    cMaxSamplingFrequency_Hz : UDINT := 2000;
    cRingBufferSizeSamples   : INT   := 64;
    cMaxZScoreAllowed        : LREAL := 6.0;
    cCompressionThresholdRLE : INT   := 3;
    cHeaderPreambleByte      : BYTE  := 16#AA;
END_VAR

// =============================================================================
// 1. SIGNAL INGESTION, OPERATOR COMMANDS & TIMERS
// =============================================================================
{region "Telemetry Engine Control and Watchdogs"}
    _fbRTrigCapture(CLK := bTriggerSnapshotLog);
    _fbRTrigClear(CLK := bClearBufferCommand);
    _fbRTrigFlush(CLK := bForceFlushToSink);
    _fbRTrigAckAnomaly(CLK := bAcknowledgeAnomalyAlarm);

    // Reset anomaly latch on operator acknowledgment
    IF _fbRTrigAckAnomaly.Q THEN
        bProcessAnomalyDetected  := FALSE;
        _bCusumDriftAlarmLatched := FALSE;
        nLoggerErrorCode         := 0;
        sDetailedLoggerStatus    := 'Anomaly alarms cleared by operator.';
END_IF

    // Purge buffer on command
    IF _fbRTrigClear.Q THEN
        M_PurgeStaleBufferSegments();
        sDetailedLoggerStatus := 'Buffer cleared by manual operator command.';
END_IF

    // Periodic heartbeat ticker
    _fbTonHeartbeatTicker(IN := NOT _fbTonHeartbeatTicker.Q, PT := tHeartbeatInterval);

    IF _fbTonHeartbeatTicker.Q AND bLoggerMasterEnable THEN
        A_UpdateDiagnosticPayload();
        A_RecalculateCompressionMetrics();
        A_SanitizeFloatingPointRegisters();
        A_SynchronizeTelemetryTimebase();
END_IF

    // Flush watchdog timer
    _fbTonFlushWatchdog(IN := (_nMasterLoggerState = 70), PT := tMaxFlushTimeout);

    IF _fbTonFlushWatchdog.Q AND NOT bBufferOverflowFault THEN
        bBufferOverflowFault  := TRUE;
        nLoggerErrorCode      := 16#A002; // Sink write timeout
        sDetailedLoggerStatus := 'FAULT: Storage sink handshake timed out during payload flush.';
        _nMasterLoggerState   := 90;     // Recovery state
END_IF
{endregion}

// =============================================================================
// 2. MASTER HIGH-DENSITY ANALYTICS SEQUENCER (10-STATE ENGINE)
// =============================================================================
CASE _nMasterLoggerState OF

    0:
        // STATE 0: IDLE STANDBY
        _sActiveLoggerPhaseName := 'STANDBY_IDLE';
        bLoggerActive           := FALSE;
        bSinkFlushInProgress    := FALSE;
        bBufferHalfFullWarning  := FALSE;
        bBufferOverflowFault    := FALSE;

        IF bLoggerMasterEnable AND NOT bBufferOverflowFault THEN
            _nMasterLoggerState     := 10; // Proceed to Ingest Sensor Channels
            bLoggerActive           := TRUE;
            sDetailedLoggerStatus   := 'Analytics logger started. Ingesting telemetry channels.';
        END_IF

    10:
        // STATE 10: INGEST & CONDITION 16 SENSOR CHANNELS
        _sActiveLoggerPhaseName := 'CHANNEL_INGESTION_RAW';

        M_IngestAndFilterChannelData(nMask := nActiveChannelBitmask, arrRawGains := arrChannelScalingGains);

        _nMasterLoggerState   := 20; // Proceed to Digital Filtering
        sDetailedLoggerStatus := 'Sensors ingested. Applying digital low-pass and Kalman filter.';

    20:
        // STATE 20: DIGITAL BUTTERWORTH & NOISE REJECTION FILTERING
        _sActiveLoggerPhaseName := 'DIGITAL_NOISE_FILTERING';

        FOR _nTempChanIdx := 1 TO 16 DO
            IF bEnableKalmanFiltering THEN
                _arrChannelFiltered[_nTempChanIdx] := M_FilterKalman1D(nChannel := _nTempChanIdx, fMeasuredZ := _arrChannelRawReadings[_nTempChanIdx]);
            ELSE
                _arrChannelFiltered[_nTempChanIdx] := (0.25 * _arrChannelRawReadings[_nTempChanIdx]) + (0.75 * _arrChannelFiltered[_nTempChanIdx]);
            END_IF
        END_FOR

        _nMasterLoggerState   := 30; // Proceed to Welford Statistical Moments
        sDetailedLoggerStatus := 'Signal filtered. Updating online statistical moments.';

    30:
        // STATE 30: STREAMING STATISTICAL MOMENTS UPDATE (WELFORD)
        _sActiveLoggerPhaseName := 'WELFORD_STATISTICAL_MOMENTS';

        M_UpdateStatisticalMomentsWelford();
        M_ComputeHigherOrderMomentsSkewKurt();

        nTotalSamplesLogged    := nTotalSamplesLogged + 1;
        nSamplesInCurrentFrame := nSamplesInCurrentFrame + 1;

        _nMasterLoggerState   := 40; // Proceed to Anomaly & Drift Detection
        sDetailedLoggerStatus := 'Moments updated. Evaluating CUSUM and Z-Score drift.';

    40:
        // STATE 40: ANOMALY & PROCESS DRIFT DETECTION (CUSUM & Z-SCORE)
        _sActiveLoggerPhaseName := 'ANOMALY_CUSUM_EVALUATION';

        _bTempAnomalyInScan := M_DetectDriftAndAnomaliesCUSUM(fZScoreLimit := fZScoreAlarmThreshold, fSlackK := fCusumSlackParameter, fDecisionH := fCusumDecisionInterval);

        IF _bTempAnomalyInScan THEN
            bProcessAnomalyDetected  := TRUE;
            _bCusumDriftAlarmLatched := TRUE;
            nActiveAnomalyCount      := nActiveAnomalyCount + 1;
            sDetailedLoggerStatus    := 'WARNING: Statistical anomaly / process drift detected!';
        END_IF

        // Decide if active frame should be compressed and serialized
        IF nSamplesInCurrentFrame >= 32 OR _fbRTrigCapture.Q THEN
            _nMasterLoggerState   := 50; // Proceed to Delta-RLE Compression
            sDetailedLoggerStatus := 'Sample batch complete. Commencing Delta-RLE compression.';
        ELSE
            _nMasterLoggerState   := 10; // Loop back for next acquisition tick
        END_IF

    50:
        // STATE 50: DELTA-RLE TELEMETRY PAYLOAD COMPRESSION
        _sActiveLoggerPhaseName := 'DELTA_RLE_COMPRESSION';

        IF bEnableRLECompression THEN
            bPayloadCompressed := M_CompressTelemetryDeltaRLE();
        ELSE
            bPayloadCompressed := FALSE;
        END_IF

        _nMasterLoggerState   := 60; // Proceed to Binary Framing & CRC32
        sDetailedLoggerStatus := 'Payload compressed. Assembling binary telemetry frame.';

    60:
        // STATE 60: BINARY TELEMETRY FRAMING & CRC32 CHECKSUM
        _sActiveLoggerPhaseName := 'BINARY_FRAME_ASSEMBLY';

        M_ConstructBinaryTelemetryFrame();
        nComputedCRC32 := M_ComputeCRC32Checksum();

        _nFrameSequenceNumber := _nFrameSequenceNumber + 1;
        _nMasterLoggerState   := 70; // Proceed to Storage Flush
        sDetailedLoggerStatus := 'Frame assembled with valid CRC32. Flushing to sink.';

    70:
        // STATE 70: ASYNCHRONOUS FLUSH TO STORAGE SINK
        _sActiveLoggerPhaseName := 'STORAGE_SINK_FLUSH';
        bSinkFlushInProgress    := TRUE;

        // Sub-controller execution for sink handshake
        _fbSinkStateController(bStart := TRUE, bStop := FALSE, bReset := FALSE, tStepTimeout := T#2S);

        IF _fbSinkStateController.eCurrentState = 90 THEN
            _fbSinkStateController(bStart := FALSE, bStop := TRUE, bReset := TRUE);
            bSinkFlushInProgress   := FALSE;
            nSamplesInCurrentFrame := 0;

            IF _nFrameSequenceNumber >= 1000 THEN
                _nMasterLoggerState   := 80; // Proceed to Partition Archive Rotation
                sDetailedLoggerStatus := 'Partition capacity reached. Rotating archive partition.';
            ELSE
                _nMasterLoggerState   := 10; // Return to channel ingestion
                sDetailedLoggerStatus := 'Frame successfully persisted to storage sink.';
            END_IF
        END_IF

    80:
        // STATE 80: PARTITION ARCHIVE ROTATION & PARTITION MIGRATION
        _sActiveLoggerPhaseName := 'PARTITION_ARCHIVE_ROTATION';

        nArchivePartitionId      := nArchivePartitionId + 1;
        _nFrameSequenceNumber    := 0;
        _sPartitionDirectoryPath := CONCAT('/var/log/telemetry/partition_', DINT_TO_STRING(nArchivePartitionId));
        _sPartitionDirectoryPath := CONCAT(_sPartitionDirectoryPath, '/');

        _nMasterLoggerState   := 10; // Return to channel ingestion
        sDetailedLoggerStatus := 'Partition rotated. Continuing telemetry acquisition.';

    90:
        // STATE 90: RECOVERY & BUFFER GARBAGE COLLECTION
        _sActiveLoggerPhaseName := 'RECOVERY_GARBAGE_COLLECTION';

        M_PurgeStaleBufferSegments();
        bSinkFlushInProgress := FALSE;

        IF _fbRTrigClear.Q OR NOT bBufferOverflowFault THEN
            _nMasterLoggerState   := 0; // Return to Standby
            sDetailedLoggerStatus := 'Recovery complete. Logger reset to standby.';
        END_IF

ELSE
    _nMasterLoggerState   := 90;
    nLoggerErrorCode      := 16#A999;
    sDetailedLoggerStatus := 'FATAL: Unknown analytics logger state index encountered.';
END_CASE

eCurrentLoggerPhase    := _nMasterLoggerState;
nActivePartitionIndex  := nArchivePartitionId;
fBufferUtilizationPct  := (TO_REAL(_fbRollingBufferPrimary.nCount) / TO_REAL(cRingBufferSizeSamples)) * 100.0;
bBufferHalfFullWarning := (fBufferUtilizationPct >= 50.0);

ACTION A_EvaluateThresholdTriggers:
// Check if any active channel exceeds physical tolerance limits
FOR _nTempChanIdx := 1 TO 16 DO
    IF ABS(_arrChannelRawReadings[_nTempChanIdx]) > 500.0 THEN
        bProcessAnomalyDetected := TRUE;
    END_IF
END_FOR
END_ACTION

ACTION A_RecalculateCompressionMetrics:
// Update throughput rate estimation
_fTempThroughputCalc     := TO_REAL(nSamplingFrequency_Hz) * 16.0 * 2.0 / 1024.0;
fEffectiveDataThroughput := _fTempThroughputCalc;
END_ACTION

ACTION A_ResetStatisticalAccumulators:
// Clear running moment accumulators
FOR _nTempChanIdx := 1 TO 16 DO
    _arrChannelMean[_nTempChanIdx]     := 0.0;
    _arrChannelM2_Accum[_nTempChanIdx] := 0.0;
    _arrChannelVariance[_nTempChanIdx] := 0.0;
    _arrChannelStdDev[_nTempChanIdx]   := 0.0;
    _arrChannelCusumPos[_nTempChanIdx] := 0.0;
    _arrChannelCusumNeg[_nTempChanIdx] := 0.0;
END_FOR
END_ACTION

